    // ===== Drive interface & supervision (VFD or actuator drive) =====
    vfdReady                     : BOOL;            // Drive ready/healthy
    vfdRunFeedback               : BOOL;            // Drive RUN feedback
    vfdFaultFeedback             : BOOL;            // Drive fault
    vfdRunFbTimeout              : TIME := T#5s;    // Timeout to receive RUN FB after start

    // ===== Drive analog feedbacks (for HMI display) =====
    vfdCurrentFeedback           : REAL;            // Current [A or %]
    vfdEngFeedback               : REAL;            // Engineering feedback (e.g., rpm, flow, etc.)
    vfdTorqueFeedback            : REAL;            // Torque (Nm or %)

    // ===== Safety (true safety inputs only) =====
    safetyOk                     : BOOL := TRUE;    // Safety chain OK
    estopOk                      : BOOL := TRUE;    // E-Stop loop OK
    guardClosedOk                : BOOL := TRUE;    // Guards/doors closed

    // ===== Interlocks (process permissives) — normal stop only =====
    interlock1                   : BOOL := TRUE;
    interlock2                   : BOOL := TRUE;
    interlock3                   : BOOL := TRUE;
    interlock4                   : BOOL := TRUE;
    interlock5                   : BOOL := TRUE;
    interlock6                   : BOOL := TRUE;

 // ===== Optional low-PV hold (normal-stop/hold) =====
    minPVEnable                  : BOOL := FALSE;   // Enable low-PV hold
    minPVTripEng                 : REAL := 0.5;     // Trip threshold (engineering units)
    minPVReleaseEng              : REAL := 0.7;     // Release threshold (engineering units)
    minPVTripTime                : TIME := T#1s;    // PV < trip for this long to trip
    minPVReleaseTime             : TIME := T#1s;    // PV > release for this long to release

    // ===== Optional high-PV hold (normal-stop/hold) =====
    maxPVEnable                  : BOOL := FALSE;   // Enable high-PV hold
    maxPVTripEng                 : REAL := 9.5;     // Trip threshold (engineering units)
    maxPVReleaseEng              : REAL := 9.2;     // Release threshold (engineering units)
    maxPVTripTime                : TIME := T#1s;    // PV > trip for this long to trip
    maxPVReleaseTime             : TIME := T#1s;    // PV < release for this long to release
	
	
END_VAR

VAR_OUTPUT
    running                      : BOOL;            // TRUE only during RUN state
    controlOutputPct             : REAL;            // Final control output 0..100%
    pidDiff                      : REAL;            // SET − ACT (post-scaling)
    pidLimited                   : BOOL;            // TRUE if saturated
    deviceState                  : STRING(80);      // Human-readable state
    vfdStartCmdOut               : BOOL;            // Asserted in Start/Run to the drive

    // ===== Holds (normal stop class) =====
    minPressureHoldActive        : BOOL;            // Low-PV hold active
    maxPressureHoldActive        : BOOL;            // High-PV hold active

    // ===== Status & HMI displays =====
    statusCode                   : INT;             // 0=Idle, 1=Running, 2=Fault
    vfdCurrentDisplay            : REAL;            // Display current [A or %]
    vfdTorqueDisplay             : REAL;            // Display torque (Nm or %)
    vfdEngDisplay                : REAL;            // Display engineering feedback (e.g., rpm)
    wirePitLevelDisplay    : REAL;            // PV (engineering units), e.g., bar/kPa/°C/…
	whiteWaterSiloLevelDisplay		: REAL;
	
END_VAR

VAR
    // ===== First scan & state/edges =====
    firstScan                    : BOOL := TRUE;    // TRUE only on first PLC cycle
	pvHoldActive  				 : BOOL;  
    step                         : INT;             // 0=Idle,10=Starting,20=Running,90=Stopping
    startOld                     : BOOL;            // Edge memory
    stopOld                      : BOOL;            // Edge memory
    rStart                       : BOOL;            // Rising edge: start
    rStop                        : BOOL;            // Rising edge: stop
    runLatch                     : BOOL;            // Toggled by Start; cleared by Stop

    // ===== Internals =====
    manualCmd                    : REAL;            // Manual command %
    yPID                         : REAL;            // PID output %
    kpUse                        : REAL;            // Kp adjusted by reverseActing

    // ===== Filtered PV (engineering units) =====
    pvEngFiltered                : REAL;

    // ===== PV & SP in % (post-scaling) =====
    pvPct                        : REAL;
    spPct                        : REAL;

    // ===== Timers =====
    tonRunFbWait                 : TON;             // Waits RUN FB after start

    // ===== Low/High PV timers =====
    tonMinPTrip                  : TON;
    tonMinPRelease               : TON;
    tonMaxPTrip                  : TON;
    tonMaxPRelease               : TON;

    // ===== Instances =====
    instPID                      : CTRL_PID;        // OSCAT PID
    instPT1                      : FT_PT1;          // PV PT1 filter

    // ===== Aggregations =====
    allSafetyOK                  : BOOL;            // safetyOk & estopOk & guardClosedOk
    anyInterlockOpen             : BOOL;            // any interlock is FALSE

    // ===== HMI display filters =====
    instPT1_TorqueDisplay        : FT_PT1;          // PT1 for torque display
    instPT1_SpeedDisplay         : FT_PT1;          // PT1 for engineering display
	
    instPT1_ProcessFeedbackEngDisplay        : FT_PT1;          // PT1 for engineering display
	instPT1_WhiteWaterSiloLevelDisplay        : FT_PT1;          // PT1 for engineering display


    processSetpointManOld        : REAL;            // Last observed manual SP (HMI)
    processSetpointAutoOld       : REAL;            // Last observed auto SP (HMI)
	minPVHoldActive: BOOL;
	maxPVHoldActive: BOOL;
END_VAR

VAR PERSISTENT
    instTUNE2AutoSetpoint        : TUNE2;           // OSCAT TUNE2 for auto SP nudge
    instTUNE2ManSetpoint         : TUNE2;           // OSCAT TUNE2 for manual output
END_VAR

VAR_IN_OUT
    // ===== Exposed setpoints =====
    processSetpointMan           : REAL;            // Manual output 0..100%
    processSetpointAuto          : REAL;            // Auto SP (engineering units or % per configuration)
END_VAR

// ============================ INITIALIZATION ============================
// Run this block only once on first cycle
IF firstScan THEN
    firstScan := FALSE;

    processSetpointMan      := instTUNE2ManSetpoint.Y;
    processSetpointManOld   := processSetpointMan;

    processSetpointAuto     := instTUNE2AutoSetpoint.Y;
    processSetpointAutoOld  := processSetpointAuto;
END_IF;


// ============================ Edges ============================
rStart := startCommand AND NOT startOld;
startOld := startCommand;

rStop  := stopCommand AND NOT stopOld;
stopOld := stopCommand;

// Start toggles run; Stop forces stop
IF rStart THEN
    runLatch := TRUE;
END_IF;
IF rStop OR stopCommand THEN
    runLatch := FALSE;
END_IF;


// ============================ Aggregations =====================
allSafetyOK := safetyOk AND estopOk AND guardClosedOk;
anyInterlockOpen := NOT (interlock1 AND interlock2 AND interlock3 AND interlock4 AND interlock5 AND interlock6);

// Defaults each cycle
vfdStartCmdOut := FALSE;


// ============================ Low/High PV HOLD supervision ============================
// LOW-PV - Hold if the wire pit level is too low
IF minPVEnable AND autoMode THEN
    tonMinPTrip   (IN := (wirePitLevel <  minPVTripEng),     PT := minPVTripTime);
    tonMinPRelease(IN := (wirePitLevel >  minPVReleaseEng),  PT := minPVReleaseTime);
    IF tonMinPTrip.Q    THEN minPVHoldActive := TRUE;  END_IF;
    IF tonMinPRelease.Q THEN minPVHoldActive := FALSE; END_IF;

ELSE
    tonMinPTrip(IN := FALSE);
    tonMinPRelease(IN := FALSE);
    minPVHoldActive := FALSE;
END_IF;

// HIGH-PV - Hold if the silo level is too high
IF maxPVEnable AND autoMode THEN
    tonMaxPTrip   (IN := (whiteWaterSiloLevel > maxPVTripEng),       PT := maxPVTripTime);
    tonMaxPRelease(IN := (whiteWaterSiloLevel < maxPVReleaseEng),    PT := maxPVReleaseTime);
    IF tonMaxPTrip.Q    THEN maxPVHoldActive := TRUE;  END_IF;
    IF tonMaxPRelease.Q THEN maxPVHoldActive := FALSE; END_IF;

ELSE
    tonMaxPTrip(IN := FALSE);
    tonMaxPRelease(IN := FALSE);
    maxPVHoldActive := FALSE;
END_IF;

// ============================ PV HOLD aggregation ============================
// NOTE: Requires pvHoldActive : BOOL in VAR section
pvHoldActive := FALSE;
IF autoMode THEN
    pvHoldActive := (minPVEnable AND minPVHoldActive) OR
                    (maxPVEnable AND maxPVHoldActive);
END_IF;


// ============================ Immediate stop / safety/fault =================
IF rStop OR stopCommand THEN
    controlOutputPct := 0.0;
    running := FALSE;
    deviceState := 'Stopping (Stop command)';
    runLatch := FALSE;
    step := 90;
END_IF;

IF vfdFaultFeedback THEN
    deviceState := 'Fault from drive';
    runLatch := FALSE;
    step := 90;
END_IF;

IF NOT allSafetyOK THEN
    deviceState := 'Stopping: safety chain open';
    runLatch := FALSE;
    step := 90;
END_IF;


// ============================ State machine =====================
CASE step OF
    // ------------------------------------------------------------
    0: // Idle
        running := FALSE;
        controlOutputPct := 0.0;
        deviceState := 'Idle';
        vfdStartCmdOut := FALSE;

        // Start request via runLatch (toggled by Start pulse)
        IF runLatch AND NOT stopCommand THEN
            // Safety must be OK; drive must be ready
            // PV hold does NOT block start anymore; it will only inhibit reference to 0%
            IF NOT allSafetyOK THEN
                deviceState := 'Start blocked: safety not OK';
                runLatch := FALSE;
                step := 0;

            ELSIF NOT vfdReady THEN
                deviceState := 'Start blocked: drive not ready';
                runLatch := FALSE;
                step := 0;

            ELSE
                IF pvHoldActive THEN
                    deviceState := 'Starting (PV hold active: output inhibited)';
                ELSE
                    deviceState := 'Starting';
                END_IF;

                vfdStartCmdOut := TRUE;                   // send START to drive
                tonRunFbWait(IN := TRUE, PT := vfdRunFbTimeout);
                step := 10;
            END_IF
        END_IF

    // ------------------------------------------------------------
    10: // Starting (await RUN feedback)
        running := FALSE;
        deviceState := 'Starting (await RUN feedback)';
        vfdStartCmdOut := TRUE;

        // If PV hold is active during start, ensure reference is inhibited to 0%
        IF pvHoldActive THEN
            controlOutputPct := 0.0;
        END_IF;

        // Safety/fault during start => stop
        IF NOT allSafetyOK THEN
            tonRunFbWait(IN := FALSE);
            deviceState := 'Stopping: safety chain open';
            vfdStartCmdOut := FALSE;
            runLatch := FALSE;
            step := 90;

        ELSIF vfdFaultFeedback THEN
            tonRunFbWait(IN := FALSE);
            deviceState := 'Fault from drive';
            vfdStartCmdOut := FALSE;
            runLatch := FALSE;
            step := 90;

        // Interlocks are normal stop only
        ELSIF anyInterlockOpen THEN
            tonRunFbWait(IN := FALSE);
            deviceState := 'Stopping: interlock open';
            vfdStartCmdOut := FALSE;
            runLatch := FALSE;
            step := 90;

        // RUN feedback arrived
        ELSIF vfdRunFeedback THEN
            tonRunFbWait(IN := FALSE);
            step := 20;

        // Timeout
        ELSIF tonRunFbWait.Q THEN
            tonRunFbWait(IN := FALSE);
            deviceState := 'Start failed: RUN feedback timeout';
            vfdStartCmdOut := FALSE;
            runLatch := FALSE;
            step := 90;
        END_IF

    // ------------------------------------------------------------
    20: // Running (control loop)
        running := TRUE;               // may be used to release other devices
        deviceState := 'Running';
        vfdStartCmdOut := TRUE;

        // Supervision
        IF NOT allSafetyOK THEN
            deviceState := 'Stopping: safety chain open';
            vfdStartCmdOut := FALSE;
            runLatch := FALSE;
            step := 90;

        ELSIF vfdFaultFeedback THEN
            deviceState := 'Fault from drive';
            vfdStartCmdOut := FALSE;
            runLatch := FALSE;
            step := 90;

        ELSIF NOT vfdReady THEN
            deviceState := 'Stopping: drive not ready';
            vfdStartCmdOut := FALSE;
            runLatch := FALSE;
            step := 90;

        ELSIF NOT vfdRunFeedback THEN
            deviceState := 'Stopping: RUN feedback lost';
            vfdStartCmdOut := FALSE;
            runLatch := FALSE;
            step := 90;

        // Interlocks → normal stop
        ELSIF anyInterlockOpen THEN
            deviceState := 'Stopping: interlock open';
            vfdStartCmdOut := FALSE;
            runLatch := FALSE;
            step := 90;

        // Start toggled OFF while running => stop
        ELSIF NOT runLatch THEN
            deviceState := 'Stopping (Start toggled off)';
            vfdStartCmdOut := FALSE;
            step := 90;

        ELSE
            // ---- Input filtering (PT1) ----
            IF enableInputFilter THEN
                instPT1(in := whiteWaterSiloLevel, T := inputFilterTime, K := inputFilterGainK, out => pvEngFiltered);
            ELSE
                pvEngFiltered := whiteWaterSiloLevel;
            END_IF

            // ---- Engineering → % scaling ----
            IF enableScaling THEN
                pvPct := _ScaleToPct(pvEngFiltered,       pLoEng, pHiEng);
                spPct := _ScaleToPct(processSetpointAuto, pLoEng, pHiEng);
            ELSE
                pvPct := pvEngFiltered;        // already %
                spPct := processSetpointAuto;  // already %
            END_IF

            // ---- Manual path (HMI) ----
            manualCmd := LIMIT(0.0, processSetpointMan, 100.0);

            // Reverse/direct action by Kp sign
            IF reverseActing THEN
                kpUse := -ABS(kp);
            ELSE
                kpUse :=  ABS(kp);
            END_IF

            // ===================== PV HOLD behavior =====================
            // When PV hold active: keep motor energized, force reference=0.0,
            // and hold PID (avoid error/windup) by forcing SET=ACT and MAN=TRUE.
            IF pvHoldActive THEN

                deviceState := 'Running (PV hold: output inhibited)';
                vfdStartCmdOut := TRUE;        // keep energized
                running := TRUE;               // keep permissives (change to FALSE if you prefer)

                instPID(
                    ACT := pvPct,
                    SET := pvPct,              // hold: SET follows PV -> DIFF ~ 0
                    M_I := 0.0,                // forced output during hold
                    MAN := TRUE,               // hold PID
                    RST := resetPID,
                    KP  := kpUse,
                    TN  := tn,
                    TV  := tv,
                    LL  := outLowLimitPct,
                    LH  := outHighLimitPct,
                    Y   => yPID,
                    DIFF=> pidDiff,
                    LIM => pidLimited
                );

                // Output inhibited to zero, motor stays enabled
                controlOutputPct := 0.0;

            ELSE
                // ===================== Normal control =====================
                instPID(
                    ACT := pvPct,
                    SET := spPct,
                    M_I := manualCmd,
                    MAN := NOT autoMode,
                    RST := resetPID,
                    KP  := kpUse,
                    TN  := tn,
                    TV  := tv,
                    LL  := outLowLimitPct,
                    LH  := outHighLimitPct,
                    Y   => yPID,
                    DIFF=> pidDiff,
                    LIM => pidLimited
                );

                // Mode select, offset, clamp
                IF autoMode THEN
                    controlOutputPct := yPID;
                ELSE
                    controlOutputPct := manualCmd;
                END_IF

                controlOutputPct := LIMIT(outLowLimitPct, controlOutputPct + outputOffsetPct, outHighLimitPct);
            END_IF
        END_IF

    // ------------------------------------------------------------
    90: // Stopping (normal, de-energize)
        running := FALSE;
        controlOutputPct := 0.0;
        vfdStartCmdOut := FALSE;
        tonRunFbWait(IN := FALSE);

        // Return to Idle once stop released and safety OK
        IF NOT stopCommand AND allSafetyOK THEN
            deviceState := 'Idle';
            step := 0;
        END_IF

    // ------------------------------------------------------------
    ELSE
        running := FALSE;
        controlOutputPct := 0.0;
        deviceState := 'Idle';
        vfdStartCmdOut := FALSE;
        step := 0;
END_CASE;


// =============================== Status code ===============================
IF vfdFaultFeedback THEN
    statusCode := 2;             // Fault
ELSIF running THEN
    statusCode := 1;             // Running
ELSE
    statusCode := 0;             // Idle
END_IF

// HMI feedbacks & status (encapsulates PT1 displays and status code if desired)
_FeedbackDisplay();

// Setpoint input handling (encapsulates TUNE2-based HMI writes & nudges)
_SetpointInputControl();

METHOD _FeedbackDisplay
VAR_INPUT
END_VAR
//instPT1_WhiteWaterSiloDisplay
//whiteWaterLevelDisplay
// 5) HMI DISPLAY SIGNALS (filtered speeds/torques + GROUP status)
instPT1_SpeedDisplay(in := vfdEngFeedback, T := displayFilterTime, K := 1.0, out => vfdEngDisplay);
instPT1_TorqueDisplay (in := vfdTorqueFeedback , T := displayFilterTime, K := 1.0, out => vfdTorqueDisplay);
instPT1_ProcessFeedbackEngDisplay(in := wirePitLevel , T := displayFilterTime, K := 1.0, out => wirePitLevelDisplay);
instPT1_WhiteWaterSiloLevelDisplay(in := whiteWaterSiloLevel , T := displayFilterTime, K := 1.0, out => whiteWaterSiloLevelDisplay);
END_METHOD

// ============================ Helper ============================
METHOD PRIVATE _ScaleToPct : REAL
VAR_INPUT
    xEng  : REAL;  // value in engineering units
    loEng : REAL;  // min eng
    hiEng : REAL;  // max eng
END_VAR
VAR
    span : REAL;
    pct  : REAL;
END_VAR

span := hiEng - loEng;
IF span = 0.0 THEN
    _ScaleToPct := 0.0; // avoid div by zero
ELSE
    pct := (xEng - loEng) / span * 100.0;
    _ScaleToPct := LIMIT(0.0, pct, 100.0);
END_IF
END_METHOD

// ============================================================================
// METHOD: _SetpointInputControl
// Purpose: Handle HMI writes for manual output using OSCAT TUNE2. Any external
//          write to manualOutputPct bigger than the configured step will pulse
//          SET for one scan. No SU/SD buttons here (PressureCtrl doesn’t use them).
// Objetivo: Tratar escrita da HMI no manualOutputPct via TUNE2. Mudança externa
//           > passo gera pulso SET de 1 varredura. Sem botões ↑/↓ neste FB.
// ============================================================================
METHOD PRIVATE _SetpointInputControl
VAR
    spManClamped : REAL;
    spAutoClamped : REAL;
	
END_VAR
// Detect external write (> step): ignore tiny jitter
IF ABS(processSetpointMan - processSetpointManOld) > instTUNE2ManSetpoint.SS THEN
    // Clamp to output limits before writing (garante limites)
    spManClamped := LIMIT(outLowLimitPct, processSetpointMan, outHighLimitPct);

    // One-scan SET pulse into TUNE2 (pulso SET de 1 ciclo)
    instTUNE2ManSetpoint(
        SET_val := spManClamped,
        SET     := TRUE
    );
    instTUNE2ManSetpoint(SET := FALSE);

    // Remember applied value (memoriza)
    processSetpointManOld := processSetpointMan;
ELSE
    // Track last seen to avoid drift (rastreia último observado)
    processSetpointManOld := processSetpointMan;
END_IF;

// Keep TUNE2 active (no SU/SD in this FB)
instTUNE2ManSetpoint(
    SET      := FALSE,
    SU       := processSetpointManInc,
    SD       := processSetpointManDec,
    RST      := FALSE,
    SS       := 0.1,           // step reference (passo de referência)
    FS       := 0.0,                     // unused
    LIMIT_L  := outLowLimitPct,
    LIMIT_H  := outHighLimitPct,
    Y        => processSetpointMan
);




// Detect external write (> step): ignore tiny jitter
IF ABS(processSetpointAuto - processSetpointAutoOld) > instTUNE2AutoSetpoint.SS THEN
    // Clamp to output limits before writing (garante limites)
    spAutoClamped := LIMIT(0, processSetpointAuto, 100);

    // One-scan SET pulse into TUNE2 (pulso SET de 1 ciclo)
    instTUNE2AutoSetpoint(
        SET_val := spAutoClamped,
        SET     := TRUE
    );
    instTUNE2AutoSetpoint(SET := FALSE);

    // Remember applied value (memoriza)
    processSetpointAutoOld := processSetpointAuto;
ELSE
    // Track last seen to avoid drift (rastreia último observado)
    processSetpointAutoOld := processSetpointAuto;
END_IF;

// Keep TUNE2 active (no SU/SD in this FB)
instTUNE2AutoSetpoint(
    SET      := FALSE,
    SU       := processSetpointAutoInc,
    SD       := processSetpointAutoDec,
    RST      := FALSE,
    SS       := 0.1,           // step reference (passo de referência)
    FS       := 0.0,                     // unused
    LIMIT_L  := 0.0,
    LIMIT_H  := 100.0,
    Y        => processSetpointAuto
);
END_METHOD

END_FUNCTION_BLOCK

// ---- Function Blocks/PaperMachine/Auxiliary/FB_ValveProcessControler.TcPOU
(*
    FB_ValveProcessControler (Simplified for Proportional Solenoid)
    Purpose: Generic process controller without VFD sequencing.
             Always evaluates the control loop (equivalent to STEP=20).
             PID (OSCAT CTRL_PID), optional reverse action, PV PT1 filter,
             engineering↔% scaling, low/high PV hold, and HMI displays.

    Status codes: statusCode INT → 0=Inhibited/Idle, 1=Running
*)

FUNCTION_BLOCK FB_ValveProcessControler
VAR_INPUT
    // ===== Manual output & Auto SP nudge =====
    processSetpointManInc        : BOOL;            // Manual output ↑ (0..100%)
    processSetpointManDec        : BOOL;            // Manual output ↓ (0..100%)
    processSetpointManSteps      : REAL := 0.1;

    processSetpointAutoInc       : BOOL;            // Auto SP ↑ (engineering units or %)
    processSetpointAutoDec       : BOOL;            // Auto SP ↓ (engineering units or %)
    processSetpointAutoSteps     : REAL := 1.0;

    // ===== Mode =====
    autoMode                     : BOOL;            // TRUE=Automatic / FALSE=Manual
    reverseActing                : BOOL := FALSE;   // TRUE: higher output decreases PV; FALSE: direct

    // ===== Process signals (PV in engineering units) =====
    processFeedbackEng           : REAL;            // PV (engineering units), e.g., bar/kPa/°C/…

    // ===== PID parameters (OSCAT CTRL_PID) =====
    kp                           : REAL := 1.0;     // Proportional gain (sign handled via reverseActing)
    tn                           : REAL := 8.0;     // Integral time [s]
    tv                           : REAL := 0.0;     // Derivative time [s]

    // ===== Output limits & offset =====
    outLowLimitPct               : REAL := 0.0;     // Min output %
    outHighLimitPct              : REAL := 100.0;   // Max output %
    outputOffsetPct              : REAL := 0.0;     // Offset added to final output

    // ===== PID housekeeping =====
    resetPID                     : BOOL;            // Reset integrator

    // ===== Input filter (OSCAT FT_PT1) =====
	deadBand					: REAL := 1.0;
    enableInputFilter            : BOOL := TRUE;    // Enable PV PT1 filter
    inputFilterTime              : TIME := T#300ms; // PT1 time constant
    inputFilterGainK             : REAL := 1.0;     // PT1 gain
    displayFilterTime            : TIME := T#20ms;  // Small PT1 for HMI displays

    // ===== Optional scaling (engineering ↔ %) =====
    enableScaling                : BOOL := TRUE;    // Enable engineering↔% scaling
    pLoEng                       : REAL := 0.0;     // Engineering low bound
    pHiEng                       : REAL := 10.0;    // Engineering high bound

    // ===== Safety (true safety inputs only) =====
    safetyOk                     : BOOL := TRUE;    // Safety chain OK
    estopOk                      : BOOL := TRUE;    // E-Stop loop OK
    guardClosedOk                : BOOL := TRUE;    // Guards/doors closed

    // ===== Interlocks (process permissives) — inhibit output =====
    interlock1                   : BOOL := TRUE;
    interlock2                   : BOOL := TRUE;
    interlock3                   : BOOL := TRUE;
    interlock4                   : BOOL := TRUE;
    interlock5                   : BOOL := TRUE;
    interlock6                   : BOOL := TRUE;

    // ===== Optional low-PV hold =====
    minPVEnable                  : BOOL := FALSE;   // Enable low-PV hold
    minPVTripEng                 : REAL := 0.5;     // Trip threshold (engineering units)
    minPVReleaseEng              : REAL := 0.7;     // Release threshold (engineering units)
    minPVTripTime                : TIME := T#1s;    // PV < trip for this long to trip
    minPVReleaseTime             : TIME := T#1s;    // PV > release for this long to release

    // ===== Optional high-PV hold =====
    maxPVEnable                  : BOOL := FALSE;   // Enable high-PV hold
    maxPVTripEng                 : REAL := 9.5;     // Trip threshold (engineering units)
    maxPVReleaseEng              : REAL := 9.2;     // Release threshold (engineering units)
    maxPVTripTime                : TIME := T#1s;    // PV > trip for this long to trip
    maxPVReleaseTime             : TIME := T#1s;    // PV < release for this long to release
END_VAR

VAR_IN_OUT
    // ===== Exposed setpoints =====
    processSetpointMan           : REAL;            // Manual output 0..100%
    processSetpointAuto          : REAL;            // Auto SP (engineering units or % per configuration)
END_VAR

VAR_OUTPUT
    running                      : BOOL;            // TRUE when permissives OK and no holds
    controlOutputPct             : REAL;            // Final control output 0..100%
    controlOutputPctDisplay             : REAL;            // Final control output 0..100%
	
    pidDiff                      : REAL;            // SET − ACT (post-scaling)
    pidLimited                   : BOOL;            // TRUE if saturated
    deviceState                  : STRING(80);      // Human-readable state

    // ===== Holds =====
    minPVHoldActive              : BOOL;            // Low-PV hold active
    maxPVHoldActive              : BOOL;            // High-PV hold active

    // ===== Status & HMI displays =====
    statusCode                   : INT;             // 0=Inhibited/Idle, 1=Running
    processFeedbackEngDisplay    : REAL;            // PV (engineering units) for HMI
END_VAR

VAR
    // ===== First scan =====
    firstScan                    : BOOL := TRUE;    // TRUE only on first PLC cycle

    // ===== Internals =====
    manualCmd                    : REAL;            // Manual command %
    yPID                         : REAL;            // PID output %
    kpUse                        : REAL;            // Kp adjusted by reverseActing

    // ===== Filtered PV (engineering units) =====
    pvEngFiltered                : REAL;

    // ===== PV & SP in % (post-scaling) =====
    pvPct                        : REAL;
    spPct                        : REAL;

    // ===== Low/High PV timers =====
    tonMinPTrip                  : TON;
    tonMinPRelease               : TON;
    tonMaxPTrip                  : TON;
    tonMaxPRelease               : TON;

    // ===== Instances =====
    instPID                      : CTRL_PID;        // OSCAT PID
    instPT1                      : FT_PT1;          // PV PT1 filter

    // ===== Aggregations =====
    allSafetyOK                  : BOOL;            // safetyOk & estopOk & guardClosedOk
    anyInterlockOpen             : BOOL;            // any interlock is FALSE

    // ===== HMI display filters =====
    instPT1_ProcessFeedbackEngDisplay : FT_PT1;     // PT1 for PV display

    // ===== TUNE2 housekeeping =====
    processSetpointManOld        : REAL;            // last observed manual SP
    processSetpointAutoOld       : REAL;            // last observed auto SP
END_VAR

VAR PERSISTENT
    instTUNE2AutoSetpoint        : TUNE2;           // OSCAT TUNE2 for auto SP nudge
    instTUNE2ManSetpoint         : TUNE2;           // OSCAT TUNE2 for manual output
END_VAR

// ============================ INITIALIZATION ============================
// Run this block only once on first cycle
IF firstScan THEN
    firstScan := FALSE;

    processSetpointMan      := instTUNE2ManSetpoint.Y;
    processSetpointManOld   := processSetpointMan;

    processSetpointAuto     := instTUNE2AutoSetpoint.Y;
    processSetpointAutoOld  := processSetpointAuto;
END_IF;



// ============================ Aggregations =====================
allSafetyOK := safetyOk AND estopOk AND guardClosedOk;
anyInterlockOpen := NOT (interlock1 AND interlock2 AND interlock3 AND interlock4 AND interlock5 AND interlock6);


// ============================ Low/High PV HOLD supervision ============================
// LOW-PV
IF minPVEnable THEN
    tonMinPTrip   (IN := (processFeedbackEng <  minPVTripEng),     PT := minPVTripTime);
    tonMinPRelease(IN := (processFeedbackEng >  minPVReleaseEng),  PT := minPVReleaseTime);
    IF tonMinPTrip.Q    THEN minPVHoldActive := TRUE;  END_IF;
    IF tonMinPRelease.Q THEN minPVHoldActive := FALSE; END_IF;

ELSE
    tonMinPTrip(IN := FALSE);
    tonMinPRelease(IN := FALSE);
    minPVHoldActive := FALSE;
END_IF;

// HIGH-PV
IF maxPVEnable THEN
    tonMaxPTrip   (IN := (processFeedbackEng > maxPVTripEng),       PT := maxPVTripTime);
    tonMaxPRelease(IN := (processFeedbackEng < maxPVReleaseEng),    PT := maxPVReleaseTime);
    IF tonMaxPTrip.Q    THEN maxPVHoldActive := TRUE;  END_IF;
    IF tonMaxPRelease.Q THEN maxPVHoldActive := FALSE; END_IF;

ELSE
    tonMaxPTrip(IN := FALSE);
    tonMaxPRelease(IN := FALSE);
    maxPVHoldActive := FALSE;
END_IF;

// ============================ Control (STEP 20 equivalent) =====================
// Default safe values
running := FALSE;
controlOutputPct := 0.0;

// Inhibit conditions (no start/stop logic — controller is "enabled" only if allowed)
IF NOT allSafetyOK THEN
    deviceState := 'Inhibited: safety chain open';

ELSIF anyInterlockOpen THEN
    deviceState := 'Inhibited: interlock open';

ELSIF (minPVEnable AND minPVHoldActive) OR (maxPVEnable AND maxPVHoldActive) THEN
    deviceState := 'Inhibited: PV hold active';

ELSE
    // Allowed to control
    running := TRUE;
    deviceState := 'Running';

    // ---- Input filtering (PT1) ----
    IF enableInputFilter THEN
        instPT1(in := processFeedbackEng, T := inputFilterTime, K := inputFilterGainK, out => pvEngFiltered);
    ELSE
        pvEngFiltered := processFeedbackEng;
    END_IF

    // ---- Engineering → % scaling ----
    IF enableScaling THEN
        pvPct := _ScaleToPct(pvEngFiltered,       pLoEng, pHiEng);
        spPct := _ScaleToPct(processSetpointAuto, pLoEng, pHiEng);
    ELSE
        pvPct := pvEngFiltered;        // already %
        spPct := processSetpointAuto;  // already %
    END_IF

    // ---- Manual path and PID with bumpless transfer ----
    manualCmd := LIMIT(0.0, processSetpointMan, 100.0);

    // Reverse/direct action by Kp sign
    IF reverseActing THEN
        kpUse := -ABS(kp);
    ELSE
        kpUse :=  ABS(kp);
    END_IF

    instPID(
        ACT := pvPct,
        SET := spPct,
        M_I := manualCmd,
        MAN := NOT autoMode,
        RST := resetPID,
        KP  := kpUse,
        TN  := tn,
        TV  := tv,
		SUP := deadBand,
        LL  := 0,
        LH  := 35,
        Y   => yPID,
        DIFF=> pidDiff,
        LIM => pidLimited
    );

    // Mode select, offset, clamp
    IF autoMode THEN
        controlOutputPct := yPID;
    ELSE
        controlOutputPct := manualCmd;
    END_IF
    controlOutputPct := LIMIT(outLowLimitPct, controlOutputPct + outputOffsetPct, outHighLimitPct);
	controlOutputPctDisplay := controlOutputPct;
END_IF;


// =============================== Status code ===============================
IF running THEN
    statusCode := 1;             // Running
ELSE
    statusCode := 0;             // Idle/Inhibited
END_IF

// HMI feedbacks & status (encapsulates PT1 displays and status code if desired)
_FeedbackDisplay();

// Setpoint input handling (encapsulates TUNE2-based HMI writes & nudges)
_SetpointInputControl();

METHOD _FeedbackDisplay
VAR_INPUT
END_VAR

instPT1_ProcessFeedbackEngDisplay(in := processFeedbackEng , T := displayFilterTime, K := 1.0, out => processFeedbackEngDisplay);
END_METHOD

// ============================ Helper ============================
METHOD PRIVATE _ScaleToPct : REAL
VAR_INPUT
    xEng  : REAL;  // value in engineering units
    loEng : REAL;  // min eng
    hiEng : REAL;  // max eng
END_VAR
VAR
    span : REAL;
    pct  : REAL;
END_VAR

span := hiEng - loEng;
IF span = 0.0 THEN
    _ScaleToPct := 0.0; // avoid div by zero
ELSE
    pct := (xEng - loEng) / span * 100.0;
    _ScaleToPct := LIMIT(0.0, pct, 100.0);
END_IF
END_METHOD

// ============================================================================
// METHOD: _SetpointInputControl
// Purpose: Handle HMI writes for manual output using OSCAT TUNE2. Any external
//          write to manualOutputPct bigger than the configured step will pulse
//          SET for one scan. No SU/SD buttons here (PressureCtrl doesn’t use them).
// Objetivo: Tratar escrita da HMI no manualOutputPct via TUNE2. Mudança externa
//           > passo gera pulso SET de 1 varredura. Sem botões ↑/↓ neste FB.
// ============================================================================
METHOD PRIVATE _SetpointInputControl
VAR
    spManClamped : REAL;
    spAutoClamped : REAL;
	
END_VAR
// Detect external write (> step): ignore tiny jitter
IF ABS(processSetpointMan - processSetpointManOld) > instTUNE2ManSetpoint.SS THEN
    // Clamp to output limits before writing (garante limites)
    spManClamped := LIMIT(outLowLimitPct, processSetpointMan, outHighLimitPct);

    // One-scan SET pulse into TUNE2 (pulso SET de 1 ciclo)
    instTUNE2ManSetpoint(
        SET_val := spManClamped,
        SET     := TRUE
    );
    instTUNE2ManSetpoint(SET := FALSE);

    // Remember applied value (memoriza)
    processSetpointManOld := processSetpointMan;
ELSE
    // Track last seen to avoid drift (rastreia último observado)
    processSetpointManOld := processSetpointMan;
END_IF;

// Keep TUNE2 active (no SU/SD in this FB)
instTUNE2ManSetpoint(
    SET      := FALSE,
    SU       := processSetpointManInc,
    SD       := processSetpointManDec,
    RST      := FALSE,
    SS       := 0.1,           // step reference (passo de referência)
    FS       := 0.0,                     // unused
    LIMIT_L  := outLowLimitPct,
    LIMIT_H  := outHighLimitPct,
    Y        => processSetpointMan
);




// Detect external write (> step): ignore tiny jitter
IF ABS(processSetpointAuto - processSetpointAutoOld) > instTUNE2AutoSetpoint.SS THEN
    // Clamp to output limits before writing (garante limites)
    spAutoClamped := LIMIT(0, processSetpointAuto, 100);

    // One-scan SET pulse into TUNE2 (pulso SET de 1 ciclo)
    instTUNE2AutoSetpoint(
        SET_val := spAutoClamped,
        SET     := TRUE
    );
    instTUNE2AutoSetpoint(SET := FALSE);

    // Remember applied value (memoriza)
    processSetpointAutoOld := processSetpointAuto;
ELSE
    // Track last seen to avoid drift (rastreia último observado)
    processSetpointAutoOld := processSetpointAuto;
END_IF;

// Keep TUNE2 active (no SU/SD in this FB)
instTUNE2AutoSetpoint(
    SET      := FALSE,
    SU       := processSetpointAutoInc,
    SD       := processSetpointAutoDec,
    RST      := FALSE,
    SS       := 0.1,           // step reference (passo de referência)
    FS       := 0.0,                     // unused
    LIMIT_L  := 0,
    LIMIT_H  := 100,
    Y        => processSetpointAuto
);
END_METHOD

END_FUNCTION_BLOCK

// ---- Function Blocks/PaperMachine/DriveControl/FB_DryingSectionDriveControl_V3.TcPOU
FUNCTION_BLOCK FB_DryingSectionDriveControl_V3
VAR_INPUT

    //==============================================================
    // GROUP INTERLOCKS & COMMANDS
    //==============================================================
    startGroup              : BOOL;  // EN: Start command (pulse) / PT: Comando de partida (pulso)
    stopGroup               : BOOL;  // EN: Stop command (level) / PT: Comando de parada (nível)

    groupFastStop           : BOOL;  // EN: Reset group faults / PT: Reset de falhas do grupo
	
    groupReset              : BOOL;  // EN: Reset group faults / PT: Reset de falhas do grupo

	
	groupNumber				: INT;
    //==============================================================
    // SPEED OFFSET / MANUAL ADJUSTMENTS
    //==============================================================
    grouSpeedDifIncCmd      : BOOL;  // EN: Lamp or indication – speed offset increasing / PT: Lâmpada ou indicação – offset de velocidade aumentando
    grouSpeedDifDecCmd      : BOOL;  // EN: Lamp or indication – speed offset decreasing / PT: Lâmpada ou indicação – offset de velocidade reduzindo
    groupRecoverSpeedCmd    : BOOL;  // EN: Recover nominal speed while TRUE / PT: Recuperar velocidade nominal enquanto TRUE

    //==============================================================
    // DRIVE STATUS INPUTS — UPPER GROUP
    //==============================================================
    upperMasterReady        : BOOL;  // EN: Upper master ready (no trip) / PT: Mestre superior pronto (sem falha)
    upperSlave1Ready        : BOOL;  // EN: Upper slave 1 ready / PT: Escravo 1 superior pronto

    //==============================================================
    // DRIVE STATUS INPUTS — LOWER GROUP
    //==============================================================
    lowerMasterReady        : BOOL;  // EN: Lower master ready (no trip) / PT: Mestre inferior pronto (sem falha)
    lowerSlave1Ready        : BOOL;  // EN: Lower slave 1 ready / PT: Escravo 1 inferior pronto

    //==============================================================
    // SPEED SETPOINTS & MODE SELECTION
    //==============================================================
    groupAutoSpeedMPM       : REAL;        // EN: Automatic mode speed [m/min] / PT: Velocidade em modo automático [m/min]
    groupManualSpeedMPM     : REAL := 50.0;// EN: Manual mode speed [m/min] / PT: Velocidade em modo manual [m/min]
    groupSpeedAutoMan       : BOOL;        // EN: Speed mode (0=Manual, 1=Auto) / PT: Modo de velocidade (0=Manual, 1=Automático)

    //==============================================================
    // SPEED & TORQUE FEEDBACKS — UPPER GROUP
    //==============================================================
    upperMasterSpeedFeedback    : REAL;  // [m/min or %]
    upperMasterTorqueFeedback   : REAL;  // [% or Nm]
    upperSlave1SpeedFeedback    : REAL;
    upperSlave1TorqueFeedback   : REAL;

    //==============================================================
    // SPEED & TORQUE FEEDBACKS — LOWER GROUP
    //==============================================================
    lowerMasterSpeedFeedback    : REAL;
    lowerMasterTorqueFeedback   : REAL;
    lowerSlave1SpeedFeedback    : REAL;
    lowerSlave1TorqueFeedback   : REAL;

    //==============================================================
    // COOLING MOTOR FAULT INPUTS
    //==============================================================
    upperMasterCoolingMotorFault : BOOL;  // EN: Upper master cooling motor fault / PT: Falha no motor de ventilação do mestre superior
    upperSlave1CoolingMotorFault : BOOL;  // EN: Upper slave 1 cooling motor fault / PT: Falha no motor de ventilação do escravo 1 superior
    lowerMasterCoolingMotorFault : BOOL;  // EN: Lower master cooling motor fault / PT: Falha no motor de ventilação do mestre inferior
    lowerSlave1CoolingMotorFault : BOOL;  // EN: Lower slave 1 cooling motor fault / PT: Falha no motor de ventilação do escravo 1 inferior

	
    lubrificationUnitFault : BOOL;  // EN: Lower slave 1 cooling motor fault / PT: Falha no motor de ventilação do escravo 1 inferior
	
	
    //==============================================================
    // FABRIC / WIRE STRETCHER ACTUATORS
    //==============================================================
    upperDryingSectionFabricStretchCmd     : BOOL;  // EN: Command to stretch upper fabric / PT: Comando para esticar a tela superior
    upperDryingSectionFabricUnstretchCmd   : BOOL;  // EN: Command to loosen upper fabric / PT: Comando para afrouxar a tela superior
	upperDryingSectionFabricStretchLimMax	: BOOL;
	upperDryingSectionFabricStretchLimMin	: BOOL;
    upperDryingSectionFabricStretcherMotorFault : BOOL;  // EN: Upper stretcher motor fault / PT: Falha no motor de estiramento superior


    lowerDryingSectionFabricStretchCmd     : BOOL;  // EN: Command to stretch lower fabric / PT: Comando para esticar a tela inferior
    lowerDryingSectionFabricUnstretchCmd   : BOOL;  // EN: Command to loosen lower fabric / PT: Comando para afrouxar a tela inferior
	lowerDryingSectionFabricStretchLimMax	: BOOL;
	lowerDryingSectionFabricStretchLimMin	: BOOL;   
 	lowerDryingSectionFabricStretcherMotorFault : BOOL;  // EN: Lower stretcher motor fault / PT: Falha no motor de estiramento inferior

    //==============================================================
    // FABRIC / WIRE OVERRUN SENSORS
    //==============================================================
    upperDryingSectionFabricOverrunOperatorSideSensor : BOOL; // EN: Upper fabric overrun sensor (operator side) / PT: Sensor de sobrecurso da tela superior (lado operador)
    upperDryingSectionFabricOverrunDriveSideSensor    : BOOL; // EN: Upper fabric overrun sensor (drive side) / PT: Sensor de sobrecurso da tela superior (lado acionamento)
    lowerDryingSectionFabricOverrunOperatorSideSensor : BOOL; // EN: Lower fabric overrun sensor (operator side) / PT: Sensor de sobrecurso da tela inferior (lado operador)
    lowerDryingSectionFabricOverrunDriveSideSensor    : BOOL; // EN: Lower fabric overrun sensor (drive side) / PT: Sensor de sobrecurso da tela inferior (lado acionamento)

    //==============================================================
    // PICK-UP ROLL POSITIONER
    //==============================================================
    pickUpRollPosCmdFwd       : BOOL;  // EN: Command forward / PT: Avanço do rolo pick-up
    pickUpRollPosCmdRev       : BOOL;  // EN: Command reverse / PT: Recuo do rolo pick-up
    pickUpRollPosLimitFwd     : BOOL;  // EN: Forward limit switch / PT: Fim de curso frontal
    pickUpRollPosLimitRev     : BOOL;  // EN: Reverse limit switch / PT: Fim de curso traseiro
    pickUpRollPosFault        : BOOL;  // EN: Positioner fault / PT: Falha no posicionador

    //==============================================================
    // SCRAPER OSCILLATORS
    //==============================================================
    babyDryerScraperOscCmd     : BOOL;  // EN: Command to start Baby Dryer scraper oscillator / PT: Comando para iniciar oscilador do Baby Dryer
    babyDryerScraperOscFault   : BOOL;  // EN: Baby Dryer oscillator fault / PT: Falha no oscilador do Baby Dryer
    babyDryerScraperOscRunning : BOOL;  // EN: Baby Dryer oscillator running / PT: Oscilador do Baby Dryer em operação

    upperGroupScraperOscCmd     : BOOL;  // EN: Upper group scraper oscillator command / PT: Comando de oscilação da raspa do grupo superior
    upperGroupScraperOscFault   : BOOL;  // EN: Upper group oscillator fault / PT: Falha no oscilador do grupo superior
    upperGroupScraperOscRunning : BOOL;  // EN: Upper group oscillator running / PT: Oscilador do grupo superior em operação

    lowerGroupScraperOscCmd     : BOOL;  // EN: Lower group scraper oscillator command / PT: Comando de oscilação da raspa do grupo inferior
    lowerGroupScraperOscFault   : BOOL;  // EN: Lower group oscillator fault / PT: Falha no oscilador do grupo inferior
    lowerGroupScraperOscRunning : BOOL;  // EN: Lower group oscillator running / PT: Oscilador do grupo inferior em operação

    //==============================================================
    // STEAM PRESSURE CONTROL (PID)
    //==============================================================
	
	paperPresenceSensor			: BOOL; //Detect if we have paper in the machine
    steamPressureAutoMan        : BOOL;  // EN: Steam pressure mode (0=Manual, 1=Auto) / PT: Modo de pressão do vapor (0=Manual, 1=Automático)
    steamPressureAutoSetpoint   : REAL;  // EN: Auto mode setpoint [bar] / PT: Setpoint em modo automático [bar]
    steamPressureManualSetpoint : REAL;  // EN: Manual mode setpoint [bar] / PT: Setpoint em modo manual [bar]
	steamPressure1 				: REAL;  // Recovery speed increment [m/min or %] (Incremento de recuperação Grupo 1)
	steamPressure2 				: REAL;  // Recovery speed increment [m/min or %] (Incremento de recuperação Grupo 1)
	
    steamPressureFeedback       : REAL;  // EN: Steam pressure feedback [bar] / PT: Retorno de pressão do vapor [bar]
    steamPressureKp             : REAL := 1.0;  // EN: PID proportional gain / PT: Ganho proporcional do PID
    steamPressureTn             : REAL := 8.0;  // EN: PID integral time [s] / PT: Tempo integral do PID [s]
    steamPressureTv             : REAL := 0.0;  // EN: PID derivative time [s] / PT: Tempo derivativo do PID [s]

	steamPressureLimLow             : REAL := 0.0;  // EN: PID proportional gain / PT: Ganho proporcional do PID
    steamPressureLimHigh             : REAL := 3.0;  // EN: PID integral time [s] / PT: Tempo integral do PID [s]

	
	
	upperMasterDiameter	: REAL := 263.878;
	upperSlave1Diameter	: REAL := 1200.980;
	lowerMasterDiameter	: REAL := 263.241;
	lowerSlave1Diameter	: REAL := 263.241;

	upperAndLowerSpeedCalibration   : REAL;  // Bias [%] between upper and lower

	
    //==============================================================
    // MACHINE CONFIGURATION STRUCT
    //==============================================================
    machineConfig               : PaperMachine_TypeHmiConfig; // EN: HMI configuration structure / PT: Estrutura de configuração da HMI

END_VAR



VAR_OUTPUT

    //==============================================================
    // STATE & DIAGNOSTICS
    //==============================================================
    deviceState                 : STRING;  // EN: Current readable device state / PT: Estado textual atual do grupo
    groupFault                  : BOOL;    // EN: Group fault active / PT: Falha ativa no grupo
    statusCode                  : INT;     // EN: 0=Idle, 1=Starting, 2=Running, 3=Fault / PT: 0=Parado, 1=Partindo, 2=Rodando, 3=Falha
	speedDif					: REAL;
	
	paperPresence				: BOOL;
    //==============================================================
    // DRIVE SPEED REFERENCES (RPM)
    //==============================================================
    upperMasterSpeedSetpointRPM : REAL;
    upperSlaveSpeedSetpointRPM  : REAL;
    lowerMasterSpeedSetpointRPM : REAL;
    lowerSlaveSpeedSetpointRPM  : REAL;


    //==============================================================
    // LINE SPEED & TORQUE REFERENCES
    //==============================================================
    nextGroupSpeedRefMPM        : REAL;  // EN: Suggested next group speed [m/min] / PT: Velocidade sugerida para o próximo grupo [m/min]

    upperSlave1TorqueRefPct     : REAL;
    upperSlave2TorqueRefPct     : REAL;
    lowerSlave1TorqueRefPct     : REAL;
    lowerSlave2TorqueRefPct     : REAL;

    //==============================================================
    // DRIVE ENABLE & RESET COMMANDS
    //==============================================================
    upperMasterEnable           : BOOL;
    upperSlave1Enable           : BOOL;
    upperMasterReset            : BOOL;
    upperSlave1Reset            : BOOL;

    lowerMasterEnable           : BOOL;
    lowerSlave1Enable           : BOOL;
    lowerMasterReset            : BOOL;
    lowerSlave1Reset            : BOOL;

    //==============================================================
    // FABRIC / WIRE STRETCHERS
    //==============================================================
    upperDryingSectionFabricStretch   : BOOL;
    upperDryingSectionFabricUnstretch : BOOL;
    lowerDryingSectionFabricStretch   : BOOL;
    lowerDryingSectionFabricUnstretch : BOOL;

    //==============================================================
    // PICK-UP ROLL POSITIONER OUTPUTS
    //==============================================================
    pickUpRollPosRunFwd          : BOOL;
    pickUpRollPosRunRev          : BOOL;

    //==============================================================
    // SCRAPER OSCILLATORS OUTPUTS
    //==============================================================
    babyDryerScraperOscRun       : BOOL;
    upperGroupScraperOscRun      : BOOL;
    lowerGroupScraperOscRun      : BOOL;

    //==============================================================
    // STEAM PRESSURE PID OUTPUT
    //==============================================================
	steamPressure : REAL; //Steam pressure display
    steamPressureControllerOutput : REAL;

    //==============================================================
    //FEEDBACKS (MPM / RPM / TOQUE)
    //==============================================================
    upperMasterSpeedMPM          : REAL;
    upperSlave1SpeedMPM          : REAL;
    lowerMasterSpeedMPM          : REAL;
    lowerSlave1SpeedMPM          : REAL;

    upperMasterSpeedRPM          : REAL;
    upperSlave1SpeedRPM          : REAL;
    lowerMasterSpeedRPM          : REAL;
    lowerSlave1SpeedRPM          : REAL;
	
    upperMasterTorque          	: REAL;
    upperSlave1Torque          	: REAL;
    lowerMasterTorque          	: REAL;
    lowerSlave1Torque          	: REAL;

    //==============================================================
    // HMI ALARMS STRUCT
    //==============================================================
    hmiAlarms                    : PaperMachine_TypeHmiAlarms;


END_VAR



VAR
    //==============================================================
    // INTERNAL FUNCTION BLOCK INSTANCES
    //==============================================================
    instFB_GroupDriveControl_V1       : FB_GroupDriveControl_V1;
    instFB_GroupSpeedControl_V1       : FB_GroupSpeedControl_V1;
    instFB_GroupDisplayFilters_V1     : FB_GroupDisplayFilters_V1;
    instFB_GroupTorqueTrimControl_V1  : FB_GroupTorqueTrimControl_V1;
    instCTRL_PID_TemperatureController: CTRL_PID;

	instFB_DryingSectionPressureControl : FB_DryingSectionPressureControl;
	
	
	

	instPT1_SteamPressureFiltered: FT_PT1;
	instFB_GroupTorqueTrimControl_V2: FB_GroupTorqueTrimControl_V2;
	upperAndLowerSpeedTrim: REAL;
	instTONGroupFaultDelay: TON;
	
    instTON_OverrunAll : TON;
    overrunAny         : BOOL;
	instTOF_PaperPresenseDelay: TOF;
	instTON_PaperPresenceSensor1: TON;
	instTON_PaperPresenceSensor2: TON;
	upperAndLowerTorqueManualEnable: BOOL;
	instFB_DryingSecSpeedControl: FB_DryingSecSpeedControl;
	instTONlubrificationUnitFaultDelay: TOn;
END_VAR



VAR PERSISTENT
    //==============================================================
    // TUNING PARAMETERS (PERSISTENT)
    //==============================================================
    instTUNE2_GroupSpeedDiference     : TUNE2; // EN: Manual tuning helper for group speed difference / PT: Auxiliar de ajuste manual da diferença de velocidade do grupo
END_VAR

// ─────────────────────────────────────────────────────────────────────────────
// MAIN CALL SEQUENCE
// ─────────────────────────────────────────────────────────────────────────────

_GroupControl();          // 1) State machine: edges, enables, stop modes

_alarmsDisplay();

_auxiliaryControls();

_SteamPressureControl();

METHOD _alarmsDisplay
VAR_INPUT
END_VAR
//==============================================================
// FABRIC OVERRUN — single TON debounce for all sensors
//==============================================================
// Any overrun sensor active (OR of all)?
overrunAny :=
    upperDryingSectionFabricOverrunOperatorSideSensor OR
    upperDryingSectionFabricOverrunDriveSideSensor    OR
    lowerDryingSectionFabricOverrunOperatorSideSensor OR
    lowerDryingSectionFabricOverrunDriveSideSensor;

// Run the single debounce timer
instTON_OverrunAll(IN := overrunAny, PT := T#5S);


//==============================================================
// ALARMS BY GROUP — set on condition; no resets here
//==============================================================
CASE groupNumber OF

    //==============================================================
    // DRYING SECTION GROUP 1 (GR1)
    //==============================================================
    1:
        //----------------------------
        // DRIVES — UPPER (GR1)
        //----------------------------
        IF NOT upperMasterReady THEN
            hmiAlarms.dryingSectionGroup1UpperMasterFaultAlarm := TRUE;
        END_IF;
        IF NOT upperSlave1Ready THEN
            hmiAlarms.dryingSectionGroup1UpperSlave1FaultAlarm := TRUE;
        END_IF;

        //----------------------------
        // COOLING MOTORS — UPPER (GR1)
        //----------------------------
        IF upperMasterCoolingMotorFault THEN
            hmiAlarms.dryingSectionGroup1UpperMasterCoolingFaultAlarm := TRUE;
        END_IF;
        IF upperSlave1CoolingMotorFault THEN
            hmiAlarms.dryingSectionGroup1UpperSlave1CoolingFaultAlarm := TRUE;
        END_IF;

        //----------------------------
        // DRIVES — LOWER (GR1)
        //----------------------------
        IF NOT lowerMasterReady THEN
            hmiAlarms.dryingSectionGroup1LowerMasterFaultAlarm := TRUE;
        END_IF;
        IF NOT lowerSlave1Ready THEN
            hmiAlarms.dryingSectionGroup1LowerSlave1FaultAlarm := TRUE;
        END_IF;


        //----------------------------
        // COOLING MOTORS — LOWER (GR1)
        //----------------------------
        IF lowerMasterCoolingMotorFault THEN
            hmiAlarms.dryingSectionGroup1LowerMasterCoolingFaultAlarm := TRUE;
        END_IF;
        IF lowerSlave1CoolingMotorFault THEN
            hmiAlarms.dryingSectionGroup1LowerSlave1CoolingFaultAlarm := TRUE;
        END_IF;

        //----------------------------
        // FABRIC OVERRUN SENSORS (GR1) — gated by TON
        //----------------------------
        IF upperDryingSectionFabricOverrunOperatorSideSensor AND instTON_OverrunAll.Q THEN
            hmiAlarms.upperDryingSectionGroup1FabricOverrunOperatorSideAlarm := TRUE;
        END_IF;
        IF upperDryingSectionFabricOverrunDriveSideSensor AND instTON_OverrunAll.Q THEN
            hmiAlarms.upperDryingSectionGroup1FabricOverrunDriveSideAlarm := TRUE;
        END_IF;
        IF lowerDryingSectionFabricOverrunOperatorSideSensor AND instTON_OverrunAll.Q THEN
            hmiAlarms.lowerDryingSectionGroup1FabricOverrunOperatorSideAlarm := TRUE;
        END_IF;
        IF lowerDryingSectionFabricOverrunDriveSideSensor AND instTON_OverrunAll.Q THEN
            hmiAlarms.lowerDryingSectionGroup1FabricOverrunDriveSideAlarm := TRUE;
        END_IF;

        //----------------------------
        // FABRIC STRETCHER MOTOR FAULTS (GR1)
        //----------------------------
        IF upperDryingSectionFabricStretcherMotorFault THEN
            hmiAlarms.upperDryingSectionGroup1FabricStretcherMotorFaultAlarm := TRUE;
        END_IF;
        IF lowerDryingSectionFabricStretcherMotorFault THEN
            hmiAlarms.lowerDryingSectionGroup1FabricStretcherMotorFaultAlarm := TRUE;
        END_IF;

        //----------------------------
        // PICK-UP ROLL POSITIONER (GR1)
        //----------------------------
        IF pickUpRollPosFault THEN
            hmiAlarms.dryingSectionGroup1PickUpRollPosFaultAlarm := TRUE;
        END_IF;

        //----------------------------
        // SCRAPER OSCILLATORS (GR1)
        //----------------------------
        IF babyDryerScraperOscFault THEN
            hmiAlarms.dryingSectionGroup1BabyDryerScraperOscFaultAlarm := TRUE;
        END_IF;
        IF upperGroupScraperOscFault THEN
            hmiAlarms.dryingSectionGroup1UpperScraperOscFaultAlarm := TRUE;
        END_IF;
        IF lowerGroupScraperOscFault THEN
            hmiAlarms.dryingSectionGroup1LowerScraperOscFaultAlarm := TRUE;
        END_IF;


    //==============================================================
    // DRYING SECTION GROUP 2 (GR2)
    //==============================================================
    2:
        //----------------------------
        // DRIVES — UPPER (GR2)
        //----------------------------
        IF NOT upperMasterReady THEN
            hmiAlarms.dryingSectionGroup2UpperMasterFaultAlarm := TRUE;
        END_IF;
        IF NOT upperSlave1Ready THEN
            hmiAlarms.dryingSectionGroup2UpperSlave1FaultAlarm := TRUE;
        END_IF;

        //----------------------------
        // COOLING MOTORS — UPPER (GR2)
        //----------------------------
        IF upperMasterCoolingMotorFault THEN
            hmiAlarms.dryingSectionGroup2UpperMasterCoolingFaultAlarm := TRUE;
        END_IF;
        IF upperSlave1CoolingMotorFault THEN
            hmiAlarms.dryingSectionGroup2UpperSlave1CoolingFaultAlarm := TRUE;
        END_IF;

        //----------------------------
        // DRIVES — LOWER (GR2)
        //----------------------------
        IF NOT lowerMasterReady THEN
            hmiAlarms.dryingSectionGroup2LowerMasterFaultAlarm := TRUE;
        END_IF;
        IF NOT lowerSlave1Ready THEN
            hmiAlarms.dryingSectionGroup2LowerSlave1FaultAlarm := TRUE;
        END_IF;

        //----------------------------
        // COOLING MOTORS — LOWER (GR2)
        //----------------------------
        IF lowerMasterCoolingMotorFault THEN
            hmiAlarms.dryingSectionGroup2LowerMasterCoolingFaultAlarm := TRUE;
        END_IF;
        IF lowerSlave1CoolingMotorFault THEN
            hmiAlarms.dryingSectionGroup2LowerSlave1CoolingFaultAlarm := TRUE;
        END_IF;

        //----------------------------
        // FABRIC OVERRUN SENSORS (GR2) — gated by TON
        //----------------------------
        IF upperDryingSectionFabricOverrunOperatorSideSensor AND instTON_OverrunAll.Q THEN
            hmiAlarms.upperDryingSectionGroup2FabricOverrunOperatorSideAlarm := TRUE;
        END_IF;
        IF upperDryingSectionFabricOverrunDriveSideSensor AND instTON_OverrunAll.Q THEN
            hmiAlarms.upperDryingSectionGroup2FabricOverrunDriveSideAlarm := TRUE;
        END_IF;
        IF lowerDryingSectionFabricOverrunOperatorSideSensor AND instTON_OverrunAll.Q THEN
            hmiAlarms.lowerDryingSectionGroup2FabricOverrunOperatorSideAlarm := TRUE;
        END_IF;
        IF lowerDryingSectionFabricOverrunDriveSideSensor AND instTON_OverrunAll.Q THEN
            hmiAlarms.lowerDryingSectionGroup2FabricOverrunDriveSideAlarm := TRUE;
        END_IF;

        //----------------------------
        // FABRIC STRETCHER MOTOR FAULTS (GR2)
        //----------------------------
        IF upperDryingSectionFabricStretcherMotorFault THEN
            hmiAlarms.upperDryingSectionGroup2FabricStretcherMotorFaultAlarm := TRUE;
        END_IF;
        IF lowerDryingSectionFabricStretcherMotorFault THEN
            hmiAlarms.lowerDryingSectionGroup2FabricStretcherMotorFaultAlarm := TRUE;
        END_IF;


    //==============================================================
    // DRYING SECTION GROUP 3 (GR3)
    //==============================================================
    3:
        //----------------------------
        // DRIVES — UPPER (GR3)
        //----------------------------
        IF NOT upperMasterReady THEN
            hmiAlarms.dryingSectionGroup3UpperMasterFaultAlarm := TRUE;
        END_IF;
        IF NOT upperSlave1Ready THEN
            hmiAlarms.dryingSectionGroup3UpperSlave1FaultAlarm := TRUE;
        END_IF;

        //----------------------------
        // COOLING MOTORS — UPPER (GR3)
        //----------------------------
        IF upperMasterCoolingMotorFault THEN
            hmiAlarms.dryingSectionGroup3UpperMasterCoolingFaultAlarm := TRUE;
        END_IF;
        IF upperSlave1CoolingMotorFault THEN
            hmiAlarms.dryingSectionGroup3UpperSlave1CoolingFaultAlarm := TRUE;
        END_IF;

        //----------------------------
        // DRIVES — LOWER (GR3)
        //----------------------------
        IF NOT lowerMasterReady THEN
            hmiAlarms.dryingSectionGroup3LowerMasterFaultAlarm := TRUE;
        END_IF;
        IF NOT lowerSlave1Ready THEN
            hmiAlarms.dryingSectionGroup3LowerSlave1FaultAlarm := TRUE;
        END_IF;


        //----------------------------
        // COOLING MOTORS — LOWER (GR3)
        //----------------------------
        IF lowerMasterCoolingMotorFault THEN
            hmiAlarms.dryingSectionGroup3LowerMasterCoolingFaultAlarm := TRUE;
        END_IF;
        IF lowerSlave1CoolingMotorFault THEN
            hmiAlarms.dryingSectionGroup3LowerSlave1CoolingFaultAlarm := TRUE;
        END_IF;

        //----------------------------
        // FABRIC OVERRUN SENSORS (GR3) — gated by TON
        //----------------------------
        IF upperDryingSectionFabricOverrunOperatorSideSensor AND instTON_OverrunAll.Q THEN
            hmiAlarms.upperDryingSectionGroup3FabricOverrunOperatorSideAlarm := TRUE;
        END_IF;
        IF upperDryingSectionFabricOverrunDriveSideSensor AND instTON_OverrunAll.Q THEN
            hmiAlarms.upperDryingSectionGroup3FabricOverrunDriveSideAlarm := TRUE;
        END_IF;
        IF lowerDryingSectionFabricOverrunOperatorSideSensor AND instTON_OverrunAll.Q THEN
            hmiAlarms.lowerDryingSectionGroup3FabricOverrunOperatorSideAlarm := TRUE;
        END_IF;
        IF lowerDryingSectionFabricOverrunDriveSideSensor AND instTON_OverrunAll.Q THEN
            hmiAlarms.lowerDryingSectionGroup3FabricOverrunDriveSideAlarm := TRUE;
        END_IF;

        //----------------------------
        // FABRIC STRETCHER MOTOR FAULTS (GR3)
        //----------------------------
        IF upperDryingSectionFabricStretcherMotorFault THEN
            hmiAlarms.upperDryingSectionGroup3FabricStretcherMotorFaultAlarm := TRUE;
        END_IF;
        IF lowerDryingSectionFabricStretcherMotorFault THEN
            hmiAlarms.lowerDryingSectionGroup3FabricStretcherMotorFaultAlarm := TRUE;
        END_IF;

ELSE
    // invalid group → do nothing (fail-safe handled below)
END_CASE;


//==============================================================
// GROUP FAULT — CURRENT GROUP (uses the HMI alarm bits)
//==============================================================
CASE groupNumber OF
    1:
        groupFault :=
            hmiAlarms.dryingSectionGroup1UpperMasterFaultAlarm OR
            hmiAlarms.dryingSectionGroup1UpperSlave1FaultAlarm OR
            hmiAlarms.dryingSectionGroup1UpperSlave2FaultAlarm OR
            hmiAlarms.dryingSectionGroup1LowerMasterFaultAlarm OR
            hmiAlarms.dryingSectionGroup1LowerSlave1FaultAlarm OR
            hmiAlarms.dryingSectionGroup1LowerSlave2FaultAlarm OR
            hmiAlarms.upperDryingSectionGroup1FabricOverrunOperatorSideAlarm OR
            hmiAlarms.upperDryingSectionGroup1FabricOverrunDriveSideAlarm OR
            hmiAlarms.lowerDryingSectionGroup1FabricOverrunOperatorSideAlarm OR
            hmiAlarms.lowerDryingSectionGroup1FabricOverrunDriveSideAlarm;

    2:
        groupFault :=
            hmiAlarms.dryingSectionGroup2UpperMasterFaultAlarm OR
            hmiAlarms.dryingSectionGroup2UpperSlave1FaultAlarm OR
            hmiAlarms.dryingSectionGroup2UpperSlave2FaultAlarm OR
            hmiAlarms.dryingSectionGroup2LowerMasterFaultAlarm OR
            hmiAlarms.dryingSectionGroup2LowerSlave1FaultAlarm OR
            hmiAlarms.dryingSectionGroup2LowerSlave2FaultAlarm OR
            hmiAlarms.upperDryingSectionGroup2FabricOverrunOperatorSideAlarm OR
            hmiAlarms.upperDryingSectionGroup2FabricOverrunDriveSideAlarm OR
            hmiAlarms.lowerDryingSectionGroup2FabricOverrunOperatorSideAlarm OR
            hmiAlarms.lowerDryingSectionGroup2FabricOverrunDriveSideAlarm;

    3:
        groupFault :=
            hmiAlarms.dryingSectionGroup3UpperMasterFaultAlarm OR
            hmiAlarms.dryingSectionGroup3UpperSlave1FaultAlarm OR
            hmiAlarms.dryingSectionGroup3UpperSlave2FaultAlarm OR
            hmiAlarms.dryingSectionGroup3LowerMasterFaultAlarm OR
            hmiAlarms.dryingSectionGroup3LowerSlave1FaultAlarm OR
            hmiAlarms.dryingSectionGroup3LowerSlave2FaultAlarm OR
            hmiAlarms.upperDryingSectionGroup3FabricOverrunOperatorSideAlarm OR
            hmiAlarms.upperDryingSectionGroup3FabricOverrunDriveSideAlarm OR
            hmiAlarms.lowerDryingSectionGroup3FabricOverrunOperatorSideAlarm OR
            hmiAlarms.lowerDryingSectionGroup3FabricOverrunDriveSideAlarm;
ELSE
    groupFault := TRUE; // fail-safe
END_CASE;

//==============================================================
// NOTE: No reset logic here. HMI reset can be added later.
//==============================================================
END_METHOD

METHOD _auxiliaryControls
VAR_INPUT
END_VAR

//-----------------------------
// UPPER FABRIC STRETCHER
//-----------------------------
// EN: Block if motor fault or limit reached
//* PT: Bloqueia se falha de motor ou fim de curso atingido */
IF NOT upperDryingSectionFabricStretcherMotorFault THEN

    // Stretch (only if not at MAX limit)
    IF upperDryingSectionFabricStretchCmd
       AND NOT upperDryingSectionFabricUnstretchCmd
       AND NOT upperDryingSectionFabricStretchLimMax THEN
        upperDryingSectionFabricStretch := TRUE;
    ELSE
        upperDryingSectionFabricStretch := FALSE;
    END_IF;

    // Unstretch (only if not at MIN limit)
    IF upperDryingSectionFabricUnstretchCmd
       AND NOT upperDryingSectionFabricStretchCmd
       AND NOT upperDryingSectionFabricStretchLimMin THEN
        upperDryingSectionFabricUnstretch := TRUE;
    ELSE
        upperDryingSectionFabricUnstretch := FALSE;
    END_IF;

ELSE
    // Fault detected → both off
    upperDryingSectionFabricStretch   := FALSE;
    upperDryingSectionFabricUnstretch := FALSE;
END_IF;


//-----------------------------
// LOWER FABRIC STRETCHER
//-----------------------------
// EN: Block if motor fault or limit reached
//* PT: Bloqueia se falha de motor ou fim de curso atingido */
IF NOT lowerDryingSectionFabricStretcherMotorFault THEN

    // Stretch (only if not at MAX limit)
    IF lowerDryingSectionFabricStretchCmd
       AND NOT lowerDryingSectionFabricUnstretchCmd
       AND NOT lowerDryingSectionFabricStretchLimMax THEN
        lowerDryingSectionFabricStretch := TRUE;
    ELSE
        lowerDryingSectionFabricStretch := FALSE;
    END_IF;

    // Unstretch (only if not at MIN limit)
    IF lowerDryingSectionFabricUnstretchCmd
       AND NOT lowerDryingSectionFabricStretchCmd
       AND NOT lowerDryingSectionFabricStretchLimMin THEN
        lowerDryingSectionFabricUnstretch := TRUE;
    ELSE
        lowerDryingSectionFabricUnstretch := FALSE;
    END_IF;

ELSE
    // Fault detected → both off
    lowerDryingSectionFabricStretch   := FALSE;
    lowerDryingSectionFabricUnstretch := FALSE;
END_IF;


//==============================================
// PICK-UP ROLL POSITIONER
//  - Uses: pickUpRollPosCmdFwd / pickUpRollPosCmdRev
//  - Safety: fault or limit reached → stop
//  - Safety (optional): if both cmds = TRUE, stop
//==============================================
IF NOT pickUpRollPosFault THEN
    // Forward
    IF pickUpRollPosCmdFwd
       AND NOT pickUpRollPosCmdRev
       AND NOT pickUpRollPosLimitFwd THEN
        // EN: run forward / PT: avança
        pickUpRollPosRunFwd := TRUE;
    ELSE
        pickUpRollPosRunFwd := FALSE;
    END_IF;

    // Reverse
    IF pickUpRollPosCmdRev
       AND NOT pickUpRollPosCmdFwd
       AND NOT pickUpRollPosLimitRev THEN
        // EN: run reverse / PT: recua
        pickUpRollPosRunRev := TRUE;
    ELSE
        pickUpRollPosRunRev := FALSE;
    END_IF;
ELSE
    // EN: Fault → stop / PT: Falha → para
    pickUpRollPosRunFwd := FALSE;
    pickUpRollPosRunRev := FALSE;
END_IF;



//==============================================
// SCRAPER OSCILLATORS
//  - Babydryer
//  - Upper group
//  - Lower group
//  - Safety: fault → stop output
//==============================================

//-----------------------------
// BABYDRYER SCRAPER OSCILLATOR
//-----------------------------
IF NOT babyDryerScraperOscFault THEN
    // EN: run only if command is active / PT: aciona somente se houver comando
    IF babyDryerScraperOscCmd AND upperMasterSpeedMPM > 10 THEN
        babyDryerScraperOscRun := TRUE;
    ELSE
        babyDryerScraperOscRun := FALSE;
    END_IF;
ELSE
    // EN: fault → force off / PT: falha → força desligado
    babyDryerScraperOscRun := FALSE;
END_IF;


//-----------------------------
// UPPER GROUP SCRAPER OSCILLATOR
//-----------------------------
IF NOT upperGroupScraperOscFault THEN
    IF upperGroupScraperOscCmd AND upperMasterSpeedMPM > 10 THEN
        upperGroupScraperOscRun := TRUE;
    ELSE
        upperGroupScraperOscRun := FALSE;
    END_IF;
ELSE
    upperGroupScraperOscRun := FALSE;
END_IF;


//-----------------------------
// LOWER GROUP SCRAPER OSCILLATOR
//-----------------------------
IF NOT lowerGroupScraperOscFault AND lowerMasterSpeedMPM > 10 THEN
    IF lowerGroupScraperOscCmd THEN
        lowerGroupScraperOscRun := TRUE;
    ELSE
        lowerGroupScraperOscRun := FALSE;
    END_IF;
ELSE
    lowerGroupScraperOscRun := FALSE;
END_IF;



//-----------------------------
// PAPER PRESENCE DISPLAY
//-----------------------------
paperPresence := paperPresenceSensor;
END_METHOD

METHOD _GroupControl
VAR_INPUT
END_VAR
(*
FUNCTION_BLOCK FB_DryingSectionDriveControl_V3
VAR_INPUT

    //==============================================================
    // GROUP INTERLOCKS & COMMANDS
    //==============================================================
    startGroup              : BOOL;  // EN: Start command (pulse) / PT: Comando de partida (pulso)
    stopGroup               : BOOL;  // EN: Stop command (level) / PT: Comando de parada (nível)
    groupReset              : BOOL;  // EN: Reset group faults / PT: Reset de falhas do grupo

    //==============================================================
    // SPEED OFFSET / MANUAL ADJUSTMENTS
    //==============================================================
    grouSpeedDifIncCmd      : BOOL;  // EN: Lamp or indication – speed offset increasing / PT: Lâmpada ou indicação – offset de velocidade aumentando
    grouSpeedDifDecCmd      : BOOL;  // EN: Lamp or indication – speed offset decreasing / PT: Lâmpada ou indicação – offset de velocidade reduzindo
    groupRecoverSpeedCmd    : BOOL;  // EN: Recover nominal speed while TRUE / PT: Recuperar velocidade nominal enquanto TRUE

    //==============================================================
    // DRIVE STATUS INPUTS — UPPER GROUP
    //==============================================================
    upperMasterReady        : BOOL;  // EN: Upper master ready (no trip) / PT: Mestre superior pronto (sem falha)
    upperSlave1Ready        : BOOL;  // EN: Upper slave 1 ready / PT: Escravo 1 superior pronto

    //==============================================================
    // DRIVE STATUS INPUTS — LOWER GROUP
    //==============================================================
    lowerMasterReady        : BOOL;  // EN: Lower master ready (no trip) / PT: Mestre inferior pronto (sem falha)
    lowerSlave1Ready        : BOOL;  // EN: Lower slave 1 ready / PT: Escravo 1 inferior pronto

    //==============================================================
    // SPEED SETPOINTS & MODE SELECTION
    //==============================================================
    groupAutoSpeedMPM       : REAL;        // EN: Automatic mode speed [m/min] / PT: Velocidade em modo automático [m/min]
    groupManualSpeedMPM     : REAL := 50.0;// EN: Manual mode speed [m/min] / PT: Velocidade em modo manual [m/min]
    groupSpeedAutoMan       : BOOL;        // EN: Speed mode (0=Manual, 1=Auto) / PT: Modo de velocidade (0=Manual, 1=Automático)

    //==============================================================
    // SPEED & TORQUE FEEDBACKS — UPPER GROUP
    //==============================================================
    upperMasterSpeedFeedback    : REAL;  // [m/min or %]
    upperMasterTorqueFeedback   : REAL;  // [% or Nm]
    upperSlave1SpeedFeedback    : REAL;
    upperSlave1TorqueFeedback   : REAL;

    //==============================================================
    // SPEED & TORQUE FEEDBACKS — LOWER GROUP
    //==============================================================
    lowerMasterSpeedFeedback    : REAL;
    lowerMasterTorqueFeedback   : REAL;
    lowerSlave1SpeedFeedback    : REAL;
    lowerSlave1TorqueFeedback   : REAL;

    //==============================================================
    // COOLING MOTOR FAULT INPUTS
    //==============================================================
    upperMasterCoolingMotorFault : BOOL;  // EN: Upper master cooling motor fault / PT: Falha no motor de ventilação do mestre superior
    upperSlave1CoolingMotorFault : BOOL;  // EN: Upper slave 1 cooling motor fault / PT: Falha no motor de ventilação do escravo 1 superior
    lowerMasterCoolingMotorFault : BOOL;  // EN: Lower master cooling motor fault / PT: Falha no motor de ventilação do mestre inferior
    lowerSlave1CoolingMotorFault : BOOL;  // EN: Lower slave 1 cooling motor fault / PT: Falha no motor de ventilação do escravo 1 inferior

    //==============================================================
    // FABRIC / WIRE STRETCHER ACTUATORS
    //==============================================================
    upperDryingSectionFabricStretchCmd     : BOOL;  // EN: Command to stretch upper fabric / PT: Comando para esticar a tela superior
    upperDryingSectionFabricUnstretchCmd   : BOOL;  // EN: Command to loosen upper fabric / PT: Comando para afrouxar a tela superior
    lowerDryingSectionFabricStretchCmd     : BOOL;  // EN: Command to stretch lower fabric / PT: Comando para esticar a tela inferior
    lowerDryingSectionFabricUnstretchCmd   : BOOL;  // EN: Command to loosen lower fabric / PT: Comando para afrouxar a tela inferior
    upperDryingSectionFabricStretcherMotorFault : BOOL;  // EN: Upper stretcher motor fault / PT: Falha no motor de estiramento superior
    lowerDryingSectionFabricStretcherMotorFault : BOOL;  // EN: Lower stretcher motor fault / PT: Falha no motor de estiramento inferior

    //==============================================================
    // FABRIC / WIRE OVERRUN SENSORS
    //==============================================================
    upperDryingSectionFabricOverrunOperatorSideSensor : BOOL; // EN: Upper fabric overrun sensor (operator side) / PT: Sensor de sobrecurso da tela superior (lado operador)
    upperDryingSectionFabricOverrunDriveSideSensor    : BOOL; // EN: Upper fabric overrun sensor (drive side) / PT: Sensor de sobrecurso da tela superior (lado acionamento)
    lowerDryingSectionFabricOverrunOperatorSideSensor : BOOL; // EN: Lower fabric overrun sensor (operator side) / PT: Sensor de sobrecurso da tela inferior (lado operador)
    lowerDryingSectionFabricOverrunDriveSideSensor    : BOOL; // EN: Lower fabric overrun sensor (drive side) / PT: Sensor de sobrecurso da tela inferior (lado acionamento)

    //==============================================================
    // PICK-UP ROLL POSITIONER
    //==============================================================
    pickUpRollPosCmdFwd       : BOOL;  // EN: Command forward / PT: Avanço do rolo pick-up
    pickUpRollPosCmdRev       : BOOL;  // EN: Command reverse / PT: Recuo do rolo pick-up
    pickUpRollPosLimitFwd     : BOOL;  // EN: Forward limit switch / PT: Fim de curso frontal
    pickUpRollPosLimitRev     : BOOL;  // EN: Reverse limit switch / PT: Fim de curso traseiro
    pickUpRollPosFault        : BOOL;  // EN: Positioner fault / PT: Falha no posicionador

    //==============================================================
    // SCRAPER OSCILLATORS
    //==============================================================
    babyDryerScraperOscCmd     : BOOL;  // EN: Command to start Baby Dryer scraper oscillator / PT: Comando para iniciar oscilador do Baby Dryer
    babyDryerScraperOscFault   : BOOL;  // EN: Baby Dryer oscillator fault / PT: Falha no oscilador do Baby Dryer
    babyDryerScraperOscRunning : BOOL;  // EN: Baby Dryer oscillator running / PT: Oscilador do Baby Dryer em operação

    upperGroupScraperOscCmd     : BOOL;  // EN: Upper group scraper oscillator command / PT: Comando de oscilação da raspa do grupo superior
    upperGroupScraperOscFault   : BOOL;  // EN: Upper group oscillator fault / PT: Falha no oscilador do grupo superior
    upperGroupScraperOscRunning : BOOL;  // EN: Upper group oscillator running / PT: Oscilador do grupo superior em operação

    lowerGroupScraperOscCmd     : BOOL;  // EN: Lower group scraper oscillator command / PT: Comando de oscilação da raspa do grupo inferior
    lowerGroupScraperOscFault   : BOOL;  // EN: Lower group oscillator fault / PT: Falha no oscilador do grupo inferior
    lowerGroupScraperOscRunning : BOOL;  // EN: Lower group oscillator running / PT: Oscilador do grupo inferior em operação

    //==============================================================
    // STEAM PRESSURE CONTROL (PID)
    //==============================================================
    steamPressureAutoMan        : BOOL;  // EN: Steam pressure mode (0=Manual, 1=Auto) / PT: Modo de pressão do vapor (0=Manual, 1=Automático)
    steamPressureAutoSetpoint   : REAL;  // EN: Auto mode setpoint [bar] / PT: Setpoint em modo automático [bar]
    steamPressureManualSetpoint : REAL;  // EN: Manual mode setpoint [bar] / PT: Setpoint em modo manual [bar]
    steamPressureFeedback       : REAL;  // EN: Steam pressure feedback [bar] / PT: Retorno de pressão do vapor [bar]
    steamPressureKp             : REAL := 1.0;  // EN: PID proportional gain / PT: Ganho proporcional do PID
    steamPressureTn             : REAL := 8.0;  // EN: PID integral time [s] / PT: Tempo integral do PID [s]
    steamPressureTv             : REAL := 0.0;  // EN: PID derivative time [s] / PT: Tempo derivativo do PID [s]

    //==============================================================
    // MACHINE CONFIGURATION STRUCT
    //==============================================================
    machineConfig               : PaperMachine_TypeHmiConfig; // EN: HMI configuration structure / PT: Estrutura de configuração da HMI

END_VAR



VAR_OUTPUT

    //==============================================================
    // STATE & DIAGNOSTICS
    //==============================================================
    deviceState                 : STRING;  // EN: Current readable device state / PT: Estado textual atual do grupo
    groupFault                  : BOOL;    // EN: Group fault active / PT: Falha ativa no grupo
    statusCode                  : INT;     // EN: 0=Idle, 1=Starting, 2=Running, 3=Fault / PT: 0=Parado, 1=Partindo, 2=Rodando, 3=Falha

    //==============================================================
    // DRIVE SPEED REFERENCES (RPM)
    //==============================================================
    upperMasterSpeedSetpointRPM : REAL;
    upperSlaveSpeedSetpointRPM  : REAL;
    lowerMasterSpeedSetpointRPM : REAL;
    lowerSlaveSpeedSetpointRPM  : REAL;


    //==============================================================
    // LINE SPEED & TORQUE REFERENCES
    //==============================================================
    nextGroupSpeedRefMPM        : REAL;  // EN: Suggested next group speed [m/min] / PT: Velocidade sugerida para o próximo grupo [m/min]

    upperSlave1TorqueRefPct     : REAL;
    upperSlave2TorqueRefPct     : REAL;
    lowerSlave1TorqueRefPct     : REAL;
    lowerSlave2TorqueRefPct     : REAL;

    //==============================================================
    // DRIVE ENABLE & RESET COMMANDS
    //==============================================================
    upperMasterEnable           : BOOL;
    upperSlave1Enable           : BOOL;
    upperMasterReset            : BOOL;
    upperSlave1Reset            : BOOL;

    lowerMasterEnable           : BOOL;
    lowerSlave1Enable           : BOOL;
    lowerMasterReset            : BOOL;
    lowerSlave1Reset            : BOOL;

    //==============================================================
    // FABRIC / WIRE STRETCHERS
    //==============================================================
    upperDryingSectionFabricStretch   : BOOL;
    upperDryingSectionFabricUnstretch : BOOL;
    lowerDryingSectionFabricStretch   : BOOL;
    lowerDryingSectionFabricUnstretch : BOOL;

    //==============================================================
    // PICK-UP ROLL POSITIONER OUTPUTS
    //==============================================================
    pickUpRollPosRunFwd          : BOOL;
    pickUpRollPosRunRev          : BOOL;

    //==============================================================
    // SCRAPER OSCILLATORS OUTPUTS
    //==============================================================
    babyDryerScraperOscRun       : BOOL;
    upperGroupScraperOscRun      : BOOL;
    lowerGroupScraperOscRun      : BOOL;

    //==============================================================
    // STEAM PRESSURE PID OUTPUT
    //==============================================================
    steamPressureControllerOutput : REAL;

    //==============================================================
    //FEEDBACKS (MPM / RPM / TOQUE)
    //==============================================================
    upperMasterSpeedMPM          : REAL;
    upperSlave1SpeedMPM          : REAL;
    lowerMasterSpeedMPM          : REAL;
    lowerSlave1SpeedMPM          : REAL;

    upperMasterSpeedRPM          : REAL;
    upperSlave1SpeedRPM          : REAL;
    lowerMasterSpeedRPM          : REAL;
    lowerSlave1SpeedRPM          : REAL;
	
    upperMasterTorque          	: REAL;
    upperSlave1Torqu          	: REAL;
    lowerMasterTorque          	: REAL;
    lowerSlave1Torque          	: REAL;

    //==============================================================
    // HMI ALARMS STRUCT
    //==============================================================
    hmiAlarms                    : PaperMachine_TypeHmiAlarms;

END_VAR



VAR
    //==============================================================
    // INTERNAL FUNCTION BLOCK INSTANCES
    //==============================================================
    instFB_GroupDriveControl_V1       : FB_GroupDriveControl_V1;
    instFB_GroupSpeedControl_V1       : FB_GroupSpeedControl_V1;
    instFB_GroupDisplayFilters_V1     : FB_GroupDisplayFilters_V1;
    instFB_GroupTorqueTrimControl_V1  : FB_GroupTorqueTrimControl_V1;
    instCTRL_PID_TemperatureController: CTRL_PID;

END_VAR



VAR PERSISTENT
    //==============================================================
    // TUNING PARAMETERS (PERSISTENT)
    //==============================================================
    instTUNE2_GroupSpeedDiference     : TUNE2; // EN: Manual tuning helper for group speed difference / PT: Auxiliar de ajuste manual da diferença de velocidade do grupo
END_VAR

	
*)
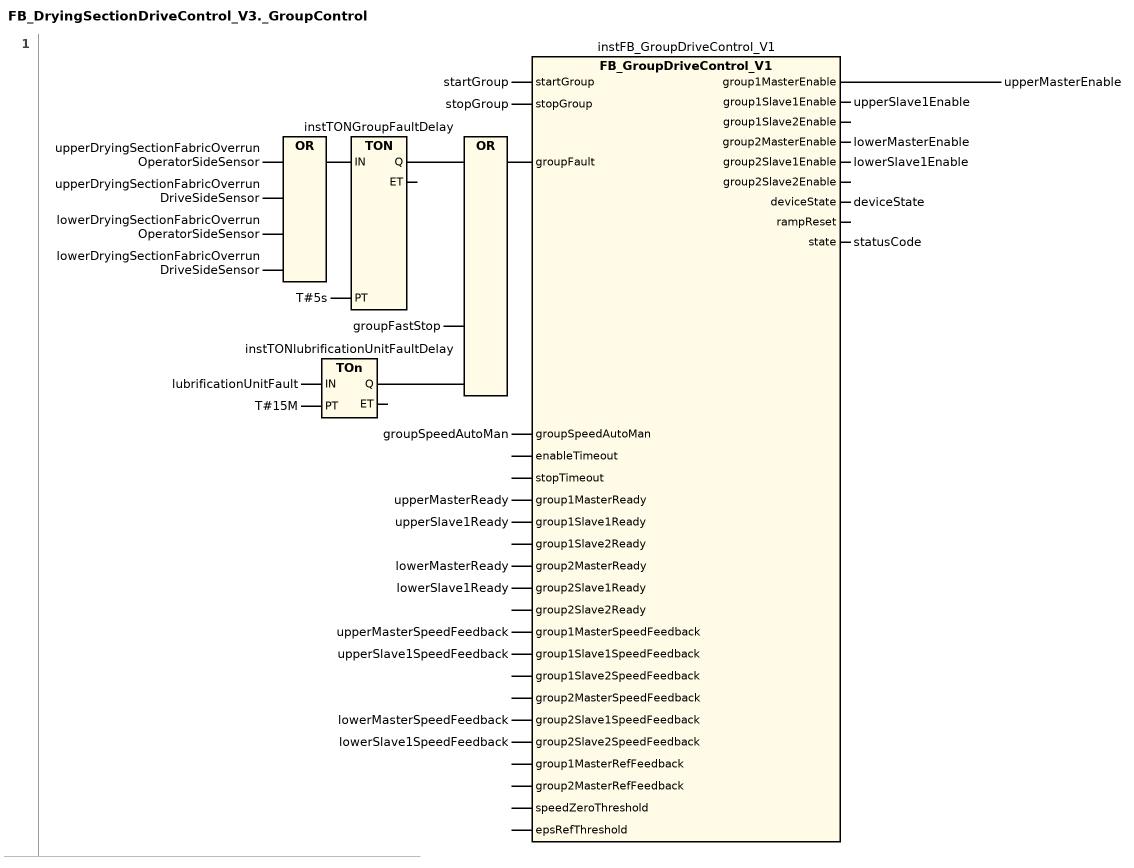
// NETWORK 1
instTONGroupFaultDelay(IN := upperDryingSectionFabricOverrunOperatorSideSensor OR upperDryingSectionFabricOverrunDriveSideSensor OR lowerDryingSectionFabricOverrunOperatorSideSensor OR lowerDryingSectionFabricOverrunDriveSideSensor, PT := T#5s); // TON
instTONlubrificationUnitFaultDelay(IN := lubrificationUnitFault, PT := T#15M); // TOn
instFB_GroupDriveControl_V1(
    startGroup := startGroup,
    stopGroup := stopGroup,
    groupFault := instTONGroupFaultDelay.Q OR groupFastStop OR instTONlubrificationUnitFaultDelay.Q,
    groupSpeedAutoMan := groupSpeedAutoMan,
    group1MasterReady := upperMasterReady,
    group1Slave1Ready := upperSlave1Ready,
    group2MasterReady := lowerMasterReady,
    group2Slave1Ready := lowerSlave1Ready,
    group1MasterSpeedFeedback := upperMasterSpeedFeedback,
    group1Slave1SpeedFeedback := upperSlave1SpeedFeedback,
    group2Slave1SpeedFeedback := lowerMasterSpeedFeedback,
    group2Slave2SpeedFeedback := lowerSlave1SpeedFeedback,
    group1Slave1Enable => upperSlave1Enable,
    group2MasterEnable => lowerMasterEnable,
    group2Slave1Enable => lowerSlave1Enable,
    deviceState => deviceState,
    state => statusCode); // FB_GroupDriveControl_V1
upperMasterEnable := instFB_GroupDriveControl_V1.group1MasterEnable;

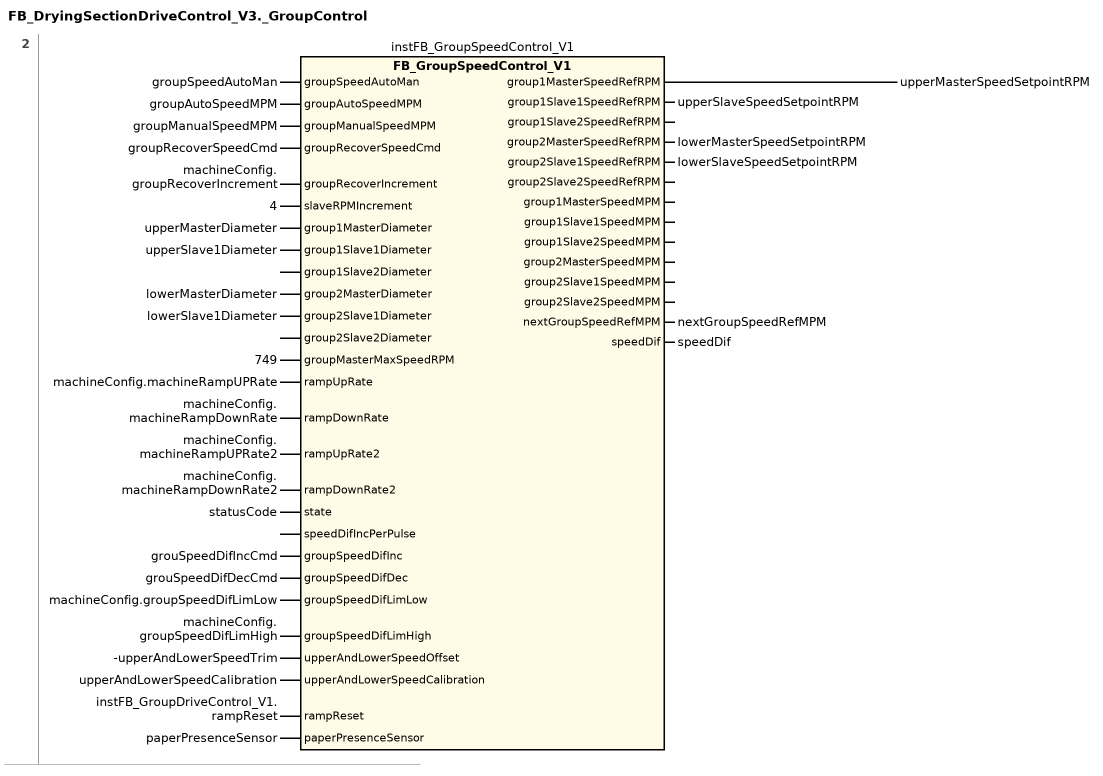
// NETWORK 2
instFB_GroupSpeedControl_V1(
    groupSpeedAutoMan := groupSpeedAutoMan,
    groupAutoSpeedMPM := groupAutoSpeedMPM,
    groupManualSpeedMPM := groupManualSpeedMPM,
    groupRecoverSpeedCmd := groupRecoverSpeedCmd,
    groupRecoverIncrement := machineConfig.groupRecoverIncrement,
    slaveRPMIncrement := 4,
    group1MasterDiameter := upperMasterDiameter,
    group1Slave1Diameter := upperSlave1Diameter,
    group2MasterDiameter := lowerMasterDiameter,
    group2Slave1Diameter := lowerSlave1Diameter,
    groupMasterMaxSpeedRPM := 749,
    rampUpRate := machineConfig.machineRampUPRate,
    rampDownRate := machineConfig.machineRampDownRate,
    rampUpRate2 := machineConfig.machineRampUPRate2,
    rampDownRate2 := machineConfig.machineRampDownRate2,
    state := statusCode,
    groupSpeedDifInc := grouSpeedDifIncCmd,
    groupSpeedDifDec := grouSpeedDifDecCmd,
    groupSpeedDifLimLow := machineConfig.groupSpeedDifLimLow,
    groupSpeedDifLimHigh := machineConfig.groupSpeedDifLimHigh,
    upperAndLowerSpeedOffset := -upperAndLowerSpeedTrim,
    upperAndLowerSpeedCalibration := upperAndLowerSpeedCalibration,
    rampReset := instFB_GroupDriveControl_V1.rampReset,
    paperPresenceSensor := paperPresenceSensor,
    group1Slave1SpeedRefRPM => upperSlaveSpeedSetpointRPM,
    group2MasterSpeedRefRPM => lowerMasterSpeedSetpointRPM,
    group2Slave1SpeedRefRPM => lowerSlaveSpeedSetpointRPM,
    nextGroupSpeedRefMPM => nextGroupSpeedRefMPM,
    speedDif => speedDif); // FB_GroupSpeedControl_V1
upperMasterSpeedSetpointRPM := instFB_GroupSpeedControl_V1.group1MasterSpeedRefRPM;

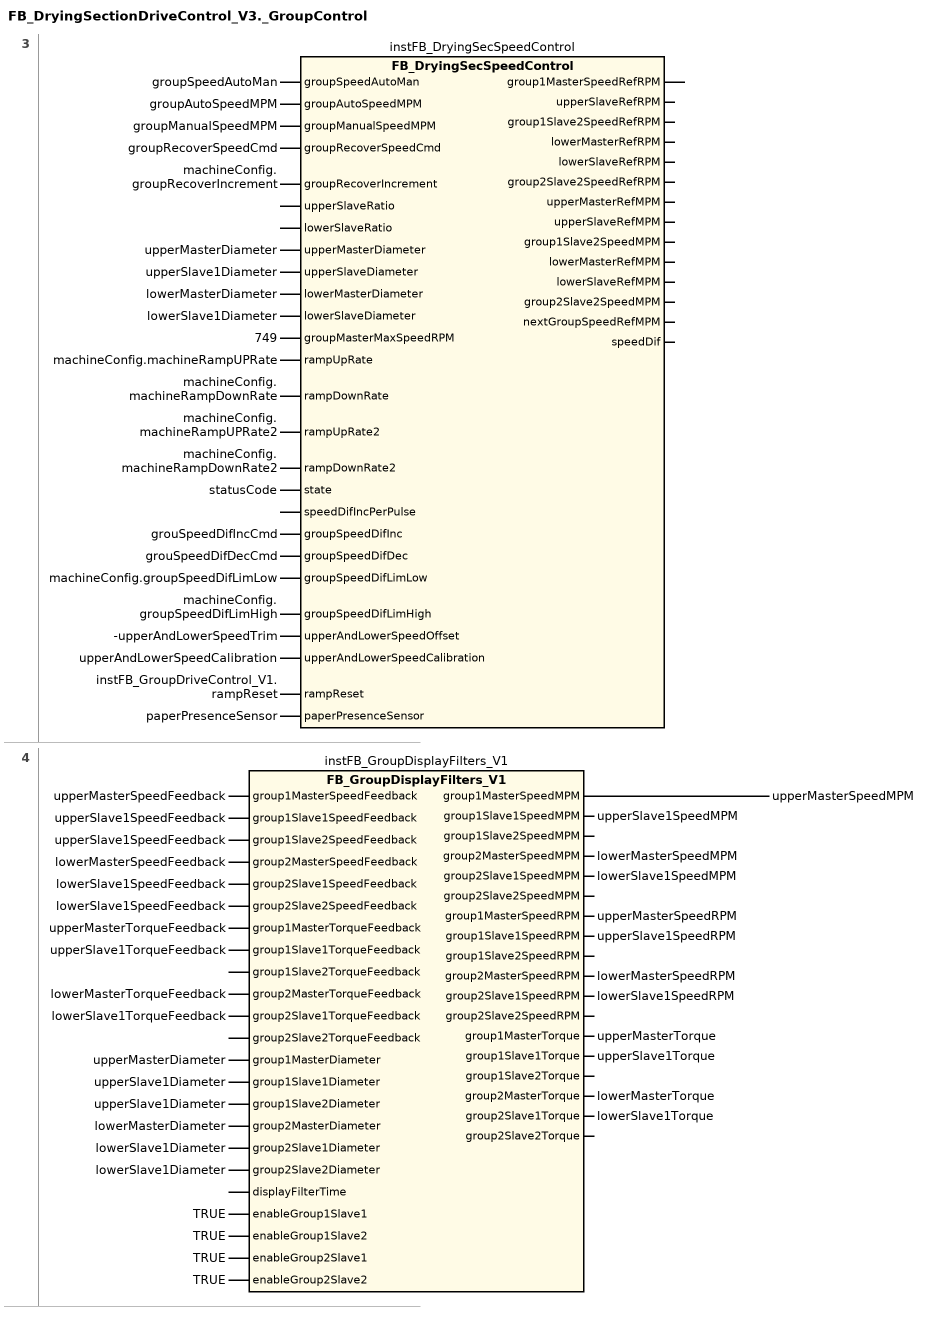
// NETWORK 3
instFB_DryingSecSpeedControl(
    groupSpeedAutoMan := groupSpeedAutoMan,
    groupAutoSpeedMPM := groupAutoSpeedMPM,
    groupManualSpeedMPM := groupManualSpeedMPM,
    groupRecoverSpeedCmd := groupRecoverSpeedCmd,
    groupRecoverIncrement := machineConfig.groupRecoverIncrement,
    upperMasterDiameter := upperMasterDiameter,
    upperSlaveDiameter := upperSlave1Diameter,
    lowerMasterDiameter := lowerMasterDiameter,
    lowerSlaveDiameter := lowerSlave1Diameter,
    groupMasterMaxSpeedRPM := 749,
    rampUpRate := machineConfig.machineRampUPRate,
    rampDownRate := machineConfig.machineRampDownRate,
    rampUpRate2 := machineConfig.machineRampUPRate2,
    rampDownRate2 := machineConfig.machineRampDownRate2,
    state := statusCode,
    groupSpeedDifInc := grouSpeedDifIncCmd,
    groupSpeedDifDec := grouSpeedDifDecCmd,
    groupSpeedDifLimLow := machineConfig.groupSpeedDifLimLow,
    groupSpeedDifLimHigh := machineConfig.groupSpeedDifLimHigh,
    upperAndLowerSpeedOffset := -upperAndLowerSpeedTrim,
    upperAndLowerSpeedCalibration := upperAndLowerSpeedCalibration,
    rampReset := instFB_GroupDriveControl_V1.rampReset,
    paperPresenceSensor := paperPresenceSensor); // FB_DryingSecSpeedControl

// NETWORK 4
instFB_GroupDisplayFilters_V1(
    group1MasterSpeedFeedback := upperMasterSpeedFeedback,
    group1Slave1SpeedFeedback := upperSlave1SpeedFeedback,
    group1Slave2SpeedFeedback := upperSlave1SpeedFeedback,
    group2MasterSpeedFeedback := lowerMasterSpeedFeedback,
    group2Slave1SpeedFeedback := lowerSlave1SpeedFeedback,
    group2Slave2SpeedFeedback := lowerSlave1SpeedFeedback,
    group1MasterTorqueFeedback := upperMasterTorqueFeedback,
    group1Slave1TorqueFeedback := upperSlave1TorqueFeedback,
    group2MasterTorqueFeedback := lowerMasterTorqueFeedback,
    group2Slave1TorqueFeedback := lowerSlave1TorqueFeedback,
    group1MasterDiameter := upperMasterDiameter,
    group1Slave1Diameter := upperSlave1Diameter,
    group1Slave2Diameter := upperSlave1Diameter,
    group2MasterDiameter := lowerMasterDiameter,
    group2Slave1Diameter := lowerSlave1Diameter,
    group2Slave2Diameter := lowerSlave1Diameter,
    enableGroup1Slave1 := TRUE,
    enableGroup1Slave2 := TRUE,
    enableGroup2Slave1 := TRUE,
    enableGroup2Slave2 := TRUE,
    group1Slave1SpeedMPM => upperSlave1SpeedMPM,
    group2MasterSpeedMPM => lowerMasterSpeedMPM,
    group2Slave1SpeedMPM => lowerSlave1SpeedMPM,
    group1MasterSpeedRPM => upperMasterSpeedRPM,
    group1Slave1SpeedRPM => upperSlave1SpeedRPM,
    group2MasterSpeedRPM => lowerMasterSpeedRPM,
    group2Slave1SpeedRPM => lowerSlave1SpeedRPM,
    group1MasterTorque => upperMasterTorque,
    group1Slave1Torque => upperSlave1Torque,
    group2MasterTorque => lowerMasterTorque,
    group2Slave1Torque => lowerSlave1Torque); // FB_GroupDisplayFilters_V1
upperMasterSpeedMPM := instFB_GroupDisplayFilters_V1.group1MasterSpeedMPM;

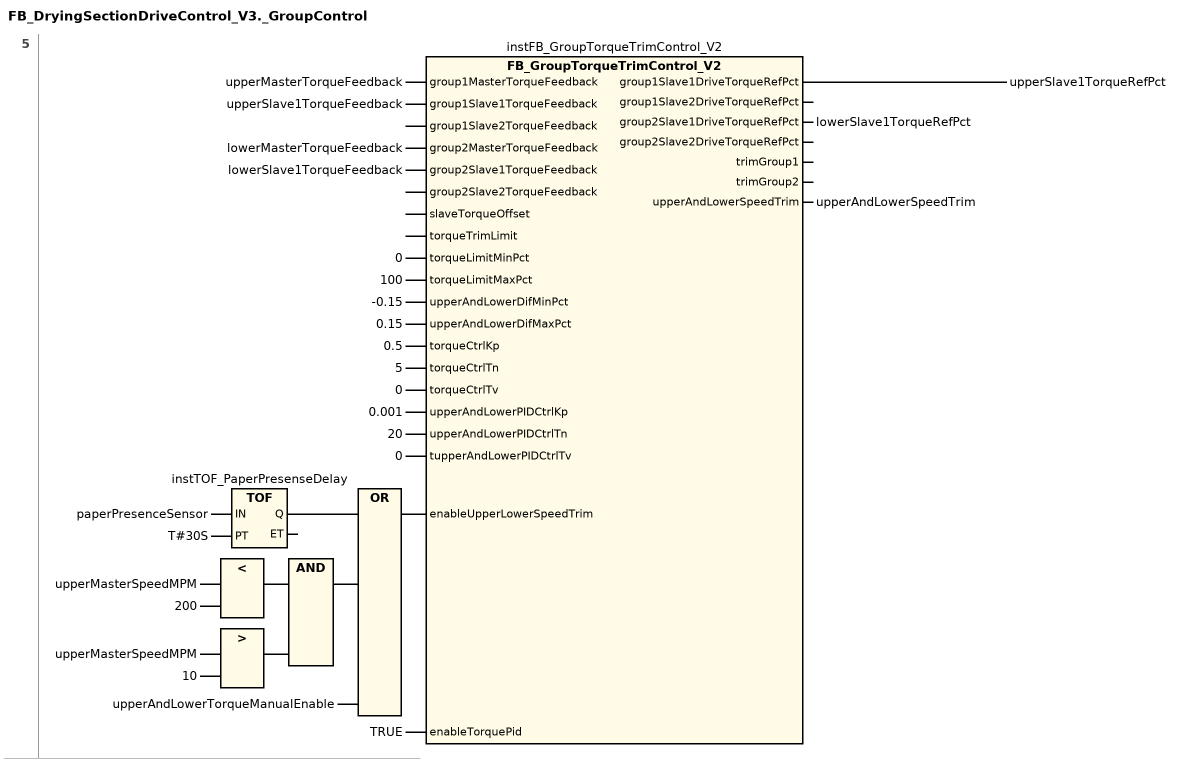
// NETWORK 5
instTOF_PaperPresenseDelay(IN := paperPresenceSensor, PT := T#30S); // TOF
instFB_GroupTorqueTrimControl_V2(
    group1MasterTorqueFeedback := upperMasterTorqueFeedback,
    group1Slave1TorqueFeedback := upperSlave1TorqueFeedback,
    group2MasterTorqueFeedback := lowerMasterTorqueFeedback,
    group2Slave1TorqueFeedback := lowerSlave1TorqueFeedback,
    torqueLimitMinPct := 0,
    torqueLimitMaxPct := 100,
    upperAndLowerDifMinPct := -0.15,
    upperAndLowerDifMaxPct := 0.15,
    torqueCtrlKp := 0.5,
    torqueCtrlTn := 5,
    torqueCtrlTv := 0,
    upperAndLowerPIDCtrlKp := 0.001,
    upperAndLowerPIDCtrlTn := 20,
    tupperAndLowerPIDCtrlTv := 0,
    enableUpperLowerSpeedTrim := instTOF_PaperPresenseDelay.Q OR upperMasterSpeedMPM < 200 AND upperMasterSpeedMPM > 10 OR upperAndLowerTorqueManualEnable,
    enableTorquePid := TRUE,
    group2Slave1DriveTorqueRefPct => lowerSlave1TorqueRefPct,
    upperAndLowerSpeedTrim => upperAndLowerSpeedTrim); // FB_GroupTorqueTrimControl_V2
upperSlave1TorqueRefPct := instFB_GroupTorqueTrimControl_V2.group1Slave1DriveTorqueRefPct;
END_METHOD

METHOD _SteamPressureControl
VAR_INPUT

END_VAR

(*
	steamPressureLimLow             : REAL := 0.0;  // EN: PID proportional gain / PT: Ganho proporcional do PID
    steamPressureLimHigh             : REAL := 3.0;  // EN: PID integral time [s] / PT: Tempo integral do PID [s]

	

*)
VAR
END_VAR
// Paper presence supervision timers
instTON_PaperPresenceSensor1(IN := NOT paperPresenceSensor, PT := T#1M);
instTON_PaperPresenceSensor2(IN := NOT paperPresenceSensor, PT := T#5M);

// Setpoint selection logic (mutually exclusive)
IF paperPresenceSensor THEN
    // Sensor enabled (ON) -> use auto setpoint
    instCTRL_PID_TemperatureController.SET := steamPressureAutoSetpoint;

ELSIF instTON_PaperPresenceSensor2.Q THEN
    // Sensor OFF for >= 5 min -> use steamPressure2
    instCTRL_PID_TemperatureController.SET := steamPressure2;

ELSIF instTON_PaperPresenceSensor1.Q AND NOT instTON_PaperPresenceSensor2.Q THEN
    // Sensor OFF for >= 1 min and < 5 min -> use steamPressure1
    instCTRL_PID_TemperatureController.SET := steamPressure1;

ELSE
    // Sensor OFF for < 1 min -> choose your desired behavior (hold last / safe default)
    // instCTRL_PID_TemperatureController.SET := steamPressureAutoSetpoint;
END_IF;



//────────────────────────────────────
// PT1 FILTER — Smooth feedback input
//────────────────────────────────────
instPT1_SteamPressureFiltered(
    in  := steamPressureFeedback,
    T   := T#1S,
    K   := 1.0,
    out => steamPressure
);

//────────────────────────────────────────────────────────────
// PID — Steam Pressure Control
//────────────────────────────────────────────────────────────
instCTRL_PID_TemperatureController(
    ACT := steamPressureFeedback,                          // Real-time feedback (PV)
//    SET := steamPressureAutoSetpoint,                 // Auto setpoint
    MAN := steamPressureAutoMan = FALSE,                   // Manual mode when AutoMan is FALSE
    M_I := steamPressureManualSetpoint,                    // Tracks manual setpoint
    RST := FALSE,                                          // No reset
    KP  := steamPressureKp,                               
    TN  := steamPressureTn,                               
    TV  := steamPressureTv,                               
    LL  := steamPressureLimLow,                                            // Output lower limit
    LH  := steamPressureLimHigh,                                          // Output upper limit [%]
    Y   => steamPressureControllerOutput                   // PID output
);
END_METHOD

END_FUNCTION_BLOCK

// ---- Function Blocks/PaperMachine/FB_DryingSecSpeedControl.TcPOU
FUNCTION_BLOCK FB_DryingSecSpeedControl
VAR_INPUT
    //==============================================================
    // ─────────────── MODE SELECTION / REFERENCES ───────────────
    //==============================================================
    groupSpeedAutoMan          : BOOL;  // TRUE = Auto, FALSE = Manual
    groupAutoSpeedMPM          : REAL;  // Auto speed reference [m/min]
    groupManualSpeedMPM        : REAL;  // Manual speed reference [m/min]
    groupRecoverSpeedCmd       : BOOL;  // Recover (temporary speed bump)
    groupRecoverIncrement      : REAL;  // Recover increment [m/min]
//    interGroupGearRatio        : REAL;  // Inter-group ratio (next section sync)

	upperSlaveRatio				: REAL := 1;
	lowerSlaveRatio				: REAL := 1;
	
    //==============================================================
    // ─────────────── DIAMETERS (mm) ───────────────
    //==============================================================
    upperMasterDiameter       : REAL;  // Diameter of group 1 master
    upperSlaveDiameter       : REAL;  // Diameter of group 1 slave 1

    lowerMasterDiameter       : REAL;  // Diameter of group 2 master
    lowerSlaveDiameter       : REAL;  // Diameter of group 2 slave 1

    //==============================================================
    // ─────────────── CONFIGURATION / LIMITS ───────────────
    //==============================================================
    groupMasterMaxSpeedRPM     : REAL;  // Max allowed master RPM
    rampUpRate					: REAL := 0.1;  // Ramp acceleration [RPM/s]
    rampDownRate				: REAL := 0.1;  // Ramp acceleration [RPM/s]
    rampUpRate2					: REAL := 0.1;  // Ramp acceleration [RPM/s]
    rampDownRate2				: REAL := 0.1;  // Ramp acceleration [RPM/s]

	
    state                      : INT;   // Machine state (5 = STOPPING)

	speedDifIncPerPulse		: REAL := 0.05;
	
    groupSpeedDifInc           : BOOL;  // Increment group speed offset
    groupSpeedDifDec           : BOOL;  // Decrement group speed offset
    groupSpeedDifLimLow        : REAL;  // Min offset [%]
    groupSpeedDifLimHigh       : REAL;  // Max offset [%]

    upperAndLowerSpeedOffset   : REAL;  // Bias [%] between group1 and group2
	upperAndLowerSpeedCalibration   : REAL;  // Bias [%] between upper and lower

    rampReset                  : BOOL;  // Reset ramp command
	
	paperPresenceSensor 		: BOOL;
	
END_VAR


VAR_OUTPUT
    //==============================================================
    // ─────────────── FINAL DRIVE SPEEDS (RPM) ───────────────
    //==============================================================
    upperMasterRefRPM    : REAL;
    upperSlaveRefRPM    : REAL;

    lowerMasterRefRPM    : REAL;
    lowerSlaveRefRPM    : REAL;


    //==============================================================
    // ─────────────── SURFACE SPEEDS (MPM) ───────────────
    //==============================================================
    upperMasterRefMPM       : REAL;
    upperSlaveRefMPM       : REAL;

    lowerMasterRefMPM       : REAL;
    lowerSlaveRefMPM       : REAL;

    //==============================================================
    // ─────────────── HANDOFF TO NEXT GROUP ───────────────
    //==============================================================
    nextGroupSpeedRefMPM       : REAL;
	speedDif					: REAL;
	
END_VAR


VAR
    //==============================================================
    // ─────────────── INTERNAL CALCULATION VARIABLES ───────────────
    //==============================================================
    masterMaxSpeedMPM          : REAL;
    baseCmdSpeedMPM            : REAL;
    cmdSpeedMPM                : REAL;
    targetRPM                  : REAL;
    rampTargetRPM              : REAL;
    baseMasterRefRPM           : REAL;
    groupSpeedOffset           : REAL;
    groupDeltaRatioAll         : REAL;
    upperLowerBiasRatio        : REAL;
    useRamp                    : BOOL;
    epsDiameter                : REAL := 0.001;

    // Gear ratios (set externally or calculated elsewhere)
    group1ToGroup1Slave1Ratio  : REAL := 1.0;
    group1ToGroup1Slave2Ratio  : REAL := 1.0;
    group1ToGroup2MasterRatio  : REAL := 1.0;
    group2ToGroup2Slave1Ratio  : REAL := 1.0;
    group2ToGroup2Slave2Ratio  : REAL := 1.0;

    // Function blocks
    instFB_Gen_SRamp           : FB_Gen_SRamp;
    instFB_SpeedDif_SRamp           : FB_Gen_SRamp;

	rampActive: BOOL;
END_VAR


VAR PERSISTENT
	
    instTUNE2_GroupSpeedDiff   : TUNE2;

END_VAR


(*

IF 	paperPresenceSensor THEN
	//slow	
	instFB_Gen_SRamp.A_UP := MAX(0.0, rampUpRate);
	instFB_Gen_SRamp.A_DN := -MAX(0.0, rampDownRate);

ELSE
	//fast
	instFB_Gen_SRamp.A_UP := MAX(0.0, rampUpRate2);
	instFB_Gen_SRamp.A_DN := -MAX(0.0, rampDownRate2);

END_IF


// Ramp function block execution
instFB_Gen_SRamp(
    X          := rampTargetRPM,
//    A_UP       := MAX(0.0, rampUpRate),
//    A_DN       := -MAX(0.0, rampDownRate),
    VU_MAX     := 1000.0,
    VD_MAX     := -1000.0,
    LIMIT_HIGH := groupMasterMaxSpeedRPM,
    RST        := rampReset);


*)

//==============================================================
// IMPLEMENTATION
//==============================================================

//====================================================================
// ═══ CALL METHOD TO CALCULATE DIAMETER RATIOS ═════════════════════
//====================================================================
_CalculateGearRatios();

